LIN {X 0,Y 509.206,Z 475.938,A -85,B 0,C 180,E1 -5494.354,E2 -5494.354} C_VEL
LIN {X 0,Y 509.283,Z 471.955,A -85,B 0,C 180,E1 -5495.543,E2 -5495.543} C_VEL
LIN {X 0,Y 509.306,Z 467.019,A -85,B 0,C 180,E1 -5496.696,E2 -5496.696} C_VEL
LIN {X 0,Y 509.468,Z 461.568,A -85,B 0,C 180,E1 -5497.73,E2 -5497.73} C_VEL
LIN {X 0,Y 509.649,Z 455.252,A -85,B 0,C 180,E1 -5498.725,E2 -5498.725} C_VEL
LIN {X 0,Y 509.834,Z 449.301,A -85,B 0,C 180,E1 -5499.521,E2 -5499.521} C_VEL
LIN {X 0,Y 509.977,Z 442.37,A -85,B 0,C 180,E1 -5500.32,E2 -5500.32} C_VEL
LIN {X 0,Y 510.292,Z 434.19,A -85,B 0,C 180,E1 -5501.117,E2 -5501.117} C_VEL
LIN {X 0,Y 510.576,Z 425.676,A -85,B 0,C 180,E1 -5501.815,E2 -5501.815} C_VEL
LIN {X 0,Y 510.837,Z 415.973,A -85,B 0,C 180,E1 -5502.474,E2 -5502.474} C_VEL
LIN {X 0,Y 511.134,Z 406.186,A -85,B 0,C 180,E1 -5503.012,E2 -5503.012} C_VEL
LIN {X 0,Y 511.34,Z 397.108,A -85,B 0,C 180,E1 -5503.411,E2 -5503.411} C_VEL
LIN {X 0,Y 511.565,Z 387.591,A -85,B 0,C 180,E1 -5503.734,E2 -5503.734} C_VEL
LIN {X 0,Y 511.759,Z 377.276,A -85,B 0,C 180,E1 -5503.982,E2 -5503.982} C_VEL
LIN {X 0,Y 512.077,Z 302.084,A -85,B 0,C 180,E1 -5505.065,E2 -5505.065} C_VEL
LIN {X 0,Y 512.113,Z 283.581,A -85,B 0,C 180,E1 -5505.327,E2 -5505.327} C_VEL
LIN {X 0,Y 510.008,Z 271.254,A -85,B 0,C 180,E1 -5505.588,E2 -5505.588} C_VEL
LIN {X 0,Y 510.017,Z 268.984,A -85,B 0,C 180,E1 -5505.998,E2 -5505.998} C_VEL
LIN {X 0,Y 510.378,Z 255.654,A -85,B 0,C 180,E1 -5508.672,E2 -5508.672} C_VEL
LIN {X 0,Y 510.735,Z 242.059,A -85,B 0,C 180,E1 -5511.386,E2 -5511.386} C_VEL
LIN {X 0,Y 511.204,Z 227.586,A -85,B 0,C 180,E1 -5514.358,E2 -5514.358} C_VEL
LIN {X 0,Y 510.607,Z 222.43,A -85,B 0,C 180,E1 -5515.475,E2 -5515.475} C_VEL
LIN {X 0,Y 509.915,Z 218.493,A -85,B 0,C 180,E1 -5516.407,E2 -5516.407} C_VEL
LIN {X 0,Y 509.86,Z 218.475,A -85,B 0,C 180,E1 -5519.751,E2 -5519.751} C_VEL
LIN {X 0,Y 509.875,Z 218.469,A -85,B 0,C 180,E1 -5522.774,E2 -5522.774} C_VEL
LIN {X 0,Y 509.828,Z 218.476,A -85,B 0,C 180,E1 -5525.578,E2 -5525.578} C_VEL
LIN {X 0,Y 509.852,Z 218.473,A -85,B 0,C 180,E1 -5528.338,E2 -5528.338} C_VEL
LIN {X 0,Y 509.857,Z 218.467,A -85,B 0,C 180,E1 -5531.425,E2 -5531.425} C_VEL
LIN {X 0,Y 509.84,Z 218.472,A -85,B 0,C 180,E1 -5534.67,E2 -5534.67} C_VEL
LIN {X 0,Y 509.835,Z 218.48,A -85,B 0,C 180,E1 -5537.51,E2 -5537.51} C_VEL
LIN {X 0,Y 509.847,Z 218.469,A -85,B 0,C 180,E1 -5540.647,E2 -5540.647} C_VEL
LIN {X 0,Y 509.825,Z 218.479,A -85,B 0,C 180,E1 -5543.646,E2 -5543.646} C_VEL
LIN {X 0,Y 509.842,Z 218.467,A -85,B 0,C 180,E1 -5546.537,E2 -5546.537} C_VEL
LIN {X 0,Y 509.843,Z 218.48,A -85,B 0,C 180,E1 -5549.334,E2 -5549.334} C_VEL
LIN {X 0,Y 509.89,Z 218.461,A -85,B 0,C 180,E1 -5552.054,E2 -5552.054} C_VEL
LIN {X 0,Y 509.876,Z 218.464,A -85,B 0,C 180,E1 -5554.704,E2 -5554.704} C_VEL
LIN {X 0,Y 509.827,Z 218.479,A -85,B 0,C 180,E1 -5557.457,E2 -5557.457} C_VEL
LIN {X 0,Y 509.917,Z 218.457,A -85,B 0,C 180,E1 -5559.844,E2 -5559.844} C_VEL
LIN {X 0,Y 509.872,Z 218.47,A -85,B 0,C 180,E1 -5563.174,E2 -5563.174} C_VEL
LIN {X 0,Y 509.863,Z 218.471,A -85,B 0,C 180,E1 -5565.634,E2 -5565.634} C_VEL
LIN {X 0,Y 509.913,Z 218.465,A -85,B 0,C 180,E1 -5568.874,E2 -5568.874} C_VEL
LIN {X 0,Y 509.921,Z 218.456,A -85,B 0,C 180,E1 -5572.078,E2 -5572.078} C_VEL
LIN {X 0,Y 509.977,Z 218.457,A -85,B 0,C 180,E1 -5574.464,E2 -5574.464} C_VEL
LIN {X 0,Y 510.055,Z 218.443,A -85,B 0,C 180,E1 -5577.63,E2 -5577.63} C_VEL
LIN {X 0,Y 510.063,Z 218.44,A -85,B 0,C 180,E1 -5580.789,E2 -5580.789} C_VEL
LIN {X 0,Y 509.952,Z 218.46,A -85,B 0,C 180,E1 -5583.16,E2 -5583.16} C_VEL
LIN {X 0,Y 509.953,Z 218.462,A -85,B 0,C 180,E1 -5586.329,E2 -5586.329} C_VEL
LIN {X 0,Y 509.914,Z 218.46,A -85,B 0,C 180,E1 -5588.72,E2 -5588.72} C_VEL
LIN {X 0,Y 509.903,Z 218.46,A -85,B 0,C 180,E1 -5591.931,E2 -5591.931} C_VEL
LIN {X 0,Y 509.892,Z 218.466,A -85,B 0,C 180,E1 -5595.241,E2 -5595.241} C_VEL
LIN {X 0,Y 509.887,Z 218.465,A -85,B 0,C 180,E1 -5598,E2 -5598} C_VEL
LIN {X 0,Y 509.848,Z 218.47,A -85,B 0,C 180,E1 -5601.001,E2 -5601.001} C_VEL
LIN {X 0,Y 509.82,Z 218.476,A -85,B 0,C 180,E1 -5603.563,E2 -5603.563} C_VEL
LIN {X 0,Y 509.908,Z 218.462,A -85,B 0,C 180,E1 -5606.378,E2 -5606.378} C_VEL
LIN {X 0,Y 509.873,Z 218.468,A -85,B 0,C 180,E1 -5608.844,E2 -5608.844} C_VEL
LIN {X 0,Y 509.819,Z 218.477,A -85,B 0,C 180,E1 -5611.59,E2 -5611.59} C_VEL
LIN {X 0,Y 509.849,Z 218.471,A -85,B 0,C 180,E1 -5614.413,E2 -5614.413} C_VEL
LIN {X 0,Y 509.816,Z 218.477,A -85,B 0,C 180,E1 -5617.34,E2 -5617.34} C_VEL
LIN {X 0,Y 509.835,Z 218.472,A -85,B 0,C 180,E1 -5620.382,E2 -5620.382} C_VEL
LIN {X 0,Y 509.836,Z 218.473,A -85,B 0,C 180,E1 -5623.064,E2 -5623.064} C_VEL
LIN {X 0,Y 509.828,Z 218.475,A -85,B 0,C 180,E1 -5625.792,E2 -5625.792} C_VEL
LIN {X 0,Y 509.862,Z 218.46,A -85,B 0,C 180,E1 -5628.575,E2 -5628.575} C_VEL
LIN {X 0,Y 509.849,Z 218.48,A -85,B 0,C 180,E1 -5631.786,E2 -5631.786} C_VEL
LIN {X 0,Y 509.827,Z 218.476,A -85,B 0,C 180,E1 -5633.737,E2 -5633.737} C_VEL
LIN {X 0,Y 509.16,Z 218.552,A -85,B 0,C 180,E1 -5634.396,E2 -5634.396} C_VEL
LIN {X 0,Y 506.343,Z 218.904,A -85,B 0,C 180,E1 -5635.468,E2 -5635.468} C_VEL
LIN {X 0,Y 503.951,Z 219.205,A -85,B 0,C 180,E1 -5636.332,E2 -5636.332} C_VEL
LIN {X 0,Y 502.903,Z 219.335,A -85,B 0,C 180,E1 -5636.998,E2 -5636.998} C_VEL
LIN {X 0,Y 502.806,Z 219.347,A -85,B 0,C 180,E1 -5637.224,E2 -5637.224} C_VEL
LIN {X 0,Y 502.811,Z 219.343,A -85,B 0,C 180,E1 -5640.065,E2 -5640.065} C_VEL
LIN {X 0,Y 502.831,Z 219.347,A -85,B 0,C 180,E1 -5642.533,E2 -5642.533} C_VEL
LIN {X 0,Y 502.823,Z 219.354,A -85,B 0,C 180,E1 -5645.299,E2 -5645.299} C_VEL
LIN {X 0,Y 502.776,Z 219.358,A -85,B 0,C 180,E1 -5647.826,E2 -5647.826} C_VEL
LIN {X 0,Y 502.822,Z 219.349,A -85,B 0,C 180,E1 -5650.4,E2 -5650.4} C_VEL
LIN {X 0,Y 502.831,Z 219.351,A -85,B 0,C 180,E1 -5652.932,E2 -5652.932} C_VEL
LIN {X 0,Y 502.848,Z 219.351,A -85,B 0,C 180,E1 -5655.429,E2 -5655.429} C_VEL
LIN {X 0,Y 502.874,Z 219.345,A -85,B 0,C 180,E1 -5658.717,E2 -5658.717} C_VEL
LIN {X 0,Y 502.899,Z 219.341,A -85,B 0,C 180,E1 -5661.967,E2 -5661.967} C_VEL
LIN {X 0,Y 502.939,Z 219.336,A -85,B 0,C 180,E1 -5664.387,E2 -5664.387} C_VEL
LIN {X 0,Y 503.023,Z 219.326,A -85,B 0,C 180,E1 -5667.598,E2 -5667.598} C_VEL
LIN {X 0,Y 503.025,Z 219.325,A -85,B 0,C 180,E1 -5670,E2 -5670} C_VEL
LIN {X 0,Y 503.023,Z 219.326,A -85,B 0,C 180,E1 -5672.402,E2 -5672.402} C_VEL
LIN {X 0,Y 502.939,Z 219.336,A -85,B 0,C 180,E1 -5675.613,E2 -5675.613} C_VEL
LIN {X 0,Y 502.899,Z 219.341,A -85,B 0,C 180,E1 -5678.033,E2 -5678.033} C_VEL
LIN {X 0,Y 502.874,Z 219.345,A -85,B 0,C 180,E1 -5681.283,E2 -5681.283} C_VEL
LIN {X 0,Y 502.848,Z 219.351,A -85,B 0,C 180,E1 -5684.571,E2 -5684.571} C_VEL
LIN {X 0,Y 502.858,Z 219.345,A -85,B 0,C 180,E1 -5687.907,E2 -5687.907} C_VEL
LIN {X 0,Y 502.825,Z 219.355,A -85,B 0,C 180,E1 -5690.536,E2 -5690.536} C_VEL
LIN {X 0,Y 502.788,Z 219.355,A -85,B 0,C 180,E1 -5693.041,E2 -5693.041} C_VEL
LIN {X 0,Y 502.836,Z 219.347,A -85,B 0,C 180,E1 -5695.676,E2 -5695.676} C_VEL
LIN {X 0,Y 502.837,Z 219.347,A -85,B 0,C 180,E1 -5698.373,E2 -5698.373} C_VEL
LIN {X 0,Y 502.793,Z 219.352,A -85,B 0,C 180,E1 -5701.5,E2 -5701.5} C_VEL
LIN {X 0,Y 502.801,Z 219.345,A -85,B 0,C 180,E1 -5704.444,E2 -5704.444} C_VEL
LIN {X 0,Y 502.778,Z 219.353,A -85,B 0,C 180,E1 -5707.179,E2 -5707.179} C_VEL
LIN {X 0,Y 502.818,Z 219.349,A -85,B 0,C 180,E1 -5710.012,E2 -5710.012} C_VEL
LIN {X 0,Y 502.77,Z 219.342,A -85,B 0,C 180,E1 -5713.231,E2 -5713.231} C_VEL
LIN {X 0,Y 502.786,Z 219.352,A -85,B 0,C 180,E1 -5715.662,E2 -5715.662} C_VEL
LIN {X 0,Y 502.83,Z 219.352,A -85,B 0,C 180,E1 -5717.865,E2 -5717.865} C_VEL
LIN {X 0,Y 502.805,Z 219.348,A -85,B 0,C 180,E1 -5721.025,E2 -5721.025} C_VEL
LIN {X 0,Y 502.78,Z 219.352,A -85,B 0,C 180,E1 -5724.168,E2 -5724.168} C_VEL
LIN {X 0,Y 502.83,Z 219.344,A -85,B 0,C 180,E1 -5726.994,E2 -5726.994} C_VEL
LIN {X 0,Y 502.812,Z 219.351,A -85,B 0,C 180,E1 -5730.065,E2 -5730.065} C_VEL
LIN {X 0,Y 502.829,Z 219.337,A -85,B 0,C 180,E1 -5732.534,E2 -5732.534} C_VEL
LIN {X 0,Y 502.783,Z 219.353,A -85,B 0,C 180,E1 -5735.31,E2 -5735.31} C_VEL
LIN {X 0,Y 502.778,Z 219.356,A -85,B 0,C 180,E1 -5737.827,E2 -5737.827} C_VEL
LIN {X 0,Y 502.823,Z 219.337,A -85,B 0,C 180,E1 -5740.401,E2 -5740.401} C_VEL
LIN {X 0,Y 502.832,Z 219.342,A -85,B 0,C 180,E1 -5742.932,E2 -5742.932} C_VEL
LIN {X 0,Y 502.85,Z 219.351,A -85,B 0,C 180,E1 -5745.43,E2 -5745.43} C_VEL
LIN {X 0,Y 502.876,Z 219.335,A -85,B 0,C 180,E1 -5748.717,E2 -5748.717} C_VEL
LIN {X 0,Y 502.901,Z 219.335,A -85,B 0,C 180,E1 -5751.967,E2 -5751.967} C_VEL
LIN {X 0,Y 502.933,Z 219.333,A -85,B 0,C 180,E1 -5754.387,E2 -5754.387} C_VEL
LIN {X 0,Y 503.025,Z 219.319,A -85,B 0,C 180,E1 -5757.598,E2 -5757.598} C_VEL
LIN {X 0,Y 503.027,Z 219.31,A -85,B 0,C 180,E1 -5760,E2 -5760} C_VEL
LIN {X 0,Y 503.024,Z 219.318,A -85,B 0,C 180,E1 -5762.403,E2 -5762.403} C_VEL
LIN {X 0,Y 502.93,Z 219.334,A -85,B 0,C 180,E1 -5765.614,E2 -5765.614} C_VEL
LIN {X 0,Y 502.864,Z 219.338,A -85,B 0,C 180,E1 -5768.844,E2 -5768.844} C_VEL
LIN {X 0,Y 502.846,Z 219.34,A -85,B 0,C 180,E1 -5772.102,E2 -5772.102} C_VEL
LIN {X 0,Y 502.849,Z 219.343,A -85,B 0,C 180,E1 -5775.4,E2 -5775.4} C_VEL
LIN {X 0,Y 502.826,Z 219.342,A -85,B 0,C 180,E1 -5778.752,E2 -5778.752} C_VEL
LIN {X 0,Y 502.783,Z 219.352,A -85,B 0,C 180,E1 -5781.312,E2 -5781.312} C_VEL
LIN {X 0,Y 502.785,Z 219.351,A -85,B 0,C 180,E1 -5783.914,E2 -5783.914} C_VEL
LIN {X 0,Y 502.865,Z 219.34,A -85,B 0,C 180,E1 -5786.566,E2 -5786.566} C_VEL
LIN {X 0,Y 502.824,Z 219.347,A -85,B 0,C 180,E1 -5789.288,E2 -5789.288} C_VEL
LIN {X 0,Y 502.782,Z 219.354,A -85,B 0,C 180,E1 -5792.085,E2 -5792.085} C_VEL
LIN {X 0,Y 502.796,Z 219.35,A -85,B 0,C 180,E1 -5794.966,E2 -5794.966} C_VEL
LIN {X 0,Y 502.794,Z 219.353,A -85,B 0,C 180,E1 -5797.954,E2 -5797.954} C_VEL
LIN {X 0,Y 502.821,Z 219.347,A -85,B 0,C 180,E1 -5801.066,E2 -5801.066} C_VEL
LIN {X 0,Y 502.787,Z 219.355,A -85,B 0,C 180,E1 -5804.53,E2 -5804.53} C_VEL
LIN {X 0,Y 502.797,Z 219.354,A -85,B 0,C 180,E1 -5807.861,E2 -5807.861} C_VEL
LIN {X 0,Y 502.804,Z 219.349,A -85,B 0,C 180,E1 -5811.024,E2 -5811.024} C_VEL
LIN {X 0,Y 502.777,Z 219.354,A -85,B 0,C 180,E1 -5814.169,E2 -5814.169} C_VEL
LIN {X 0,Y 502.835,Z 219.345,A -85,B 0,C 180,E1 -5816.994,E2 -5816.994} C_VEL
LIN {X 0,Y 502.817,Z 219.352,A -85,B 0,C 180,E1 -5820.065,E2 -5820.065} C_VEL
LIN {X 0,Y 502.878,Z 219.516,A -85,B 0,C 180,E1 -5823.479,E2 -5823.479} C_VEL
LIN {X 0,Y 504.2,Z 227.447,A -85,B 0,C 180,E1 -5825.281,E2 -5825.281} C_VEL
LIN {X 0,Y 503.846,Z 238.784,A -85,B 0,C 180,E1 -5827.66,E2 -5827.66} C_VEL
LIN {X 0,Y 503.534,Z 251.309,A -85,B 0,C 180,E1 -5830.217,E2 -5830.217} C_VEL
LIN {X 0,Y 503.109,Z 265.765,A -85,B 0,C 180,E1 -5833.151,E2 -5833.151} C_VEL
LIN {X 0,Y 502.954,Z 270.794,A -85,B 0,C 180,E1 -5834.165,E2 -5834.165} C_VEL
LIN {X 0,Y 503.729,Z 275.59,A -85,B 0,C 180,E1 -5834.3,E2 -5834.3} C_VEL
LIN {X 0,Y 505.349,Z 285.243,A -85,B 0,C 180,E1 -5834.49,E2 -5834.49} C_VEL
LIN {X 0,Y 504.877,Z 375.752,A -85,B 0,C 180,E1 -5835.798,E2 -5835.798} C_VEL
LIN {X 0,Y 504.677,Z 386.523,A -85,B 0,C 180,E1 -5836.049,E2 -5836.049} C_VEL
LIN {X 0,Y 504.465,Z 395.627,A -85,B 0,C 180,E1 -5836.351,E2 -5836.351} C_VEL
LIN {X 0,Y 504.192,Z 405.993,A -85,B 0,C 180,E1 -5836.806,E2 -5836.806} C_VEL
LIN {X 0,Y 503.889,Z 415.953,A -85,B 0,C 180,E1 -5837.362,E2 -5837.362} C_VEL
LIN {X 0,Y 503.605,Z 424.129,A -85,B 0,C 180,E1 -5837.917,E2 -5837.917} C_VEL
LIN {X 0,Y 503.336,Z 432.861,A -85,B 0,C 180,E1 -5838.625,E2 -5838.625} C_VEL
LIN {X 0,Y 503.048,Z 440.257,A -85,B 0,C 180,E1 -5839.332,E2 -5839.332} C_VEL
LIN {X 0,Y 502.842,Z 447.479,A -85,B 0,C 180,E1 -5840.142,E2 -5840.142} C_VEL
LIN {X 0,Y 502.642,Z 453.682,A -85,B 0,C 180,E1 -5840.95,E2 -5840.95} C_VEL
LIN {X 0,Y 502.437,Z 460.219,A -85,B 0,C 180,E1 -5841.959,E2 -5841.959} C_VEL
LIN {X 0,Y 502.275,Z 465.773,A -85,B 0,C 180,E1 -5842.988,E2 -5842.988} C_VEL
LIN {X 0,Y 502.201,Z 470.209,A -85,B 0,C 180,E1 -5843.975,E2 -5843.975} C_VEL
LIN {X 0,Y 502.112,Z 474.529,A -85,B 0,C 180,E1 -5845.183,E2 -5845.183} C_VEL
LIN {X 0,Y 502.139,Z 476.894,A -85,B 0,C 180,E1 -5845.987,E2 -5845.987} C_VEL
LIN {X 0,Y 502.12,Z 478.689,A -85,B 0,C 180,E1 -5846.791,E2 -5846.791} C_VEL
LIN {X 0,Y 502.037,Z 481.127,A -85,B 0,C 180,E1 -5848.396,E2 -5848.396} C_VEL
LIN {X 0,Y 501.991,Z 481.713,A -85,B 0,C 180,E1 -5849.198,E2 -5849.198} C_VEL
LIN {X 0,Y 501.991,Z 481.713,A -85,B 0,C 180,E1 -5850.802,E2 -5850.802} C_VEL
LIN {X 0,Y 502.037,Z 481.127,A -85,B 0,C 180,E1 -5851.604,E2 -5851.604} C_VEL
LIN {X 0,Y 502.12,Z 478.689,A -85,B 0,C 180,E1 -5853.209,E2 -5853.209} C_VEL
LIN {X 0,Y 502.105,Z 475.744,A -85,B 0,C 180,E1 -5854.415,E2 -5854.415} C_VEL
LIN {X 0,Y 502.199,Z 471.762,A -85,B 0,C 180,E1 -5855.622,E2 -5855.622} C_VEL
LIN {X 0,Y 502.219,Z 466.825,A -85,B 0,C 180,E1 -5856.791,E2 -5856.791} C_VEL
LIN {X 0,Y 502.393,Z 461.374,A -85,B 0,C 180,E1 -5857.839,E2 -5857.839} C_VEL
LIN {X 0,Y 502.59,Z 455.058,A -85,B 0,C 180,E1 -5858.848,E2 -5858.848} C_VEL
LIN {X 0,Y 502.796,Z 449.107,A -85,B 0,C 180,E1 -5859.656,E2 -5859.656} C_VEL
LIN {X 0,Y 502.954,Z 442.176,A -85,B 0,C 180,E1 -5860.466,E2 -5860.466} C_VEL
LIN {X 0,Y 503.289,Z 433.996,A -85,B 0,C 180,E1 -5861.274,E2 -5861.274} C_VEL
LIN {X 0,Y 503.601,Z 425.482,A -85,B 0,C 180,E1 -5861.981,E2 -5861.981} C_VEL
LIN {X 0,Y 503.869,Z 416.244,A -85,B 0,C 180,E1 -5862.62,E2 -5862.62} C_VEL
LIN {X 0,Y 504.182,Z 407,A -85,B 0,C 180,E1 -5863.143,E2 -5863.143} C_VEL
LIN {X 0,Y 504.423,Z 396.915,A -85,B 0,C 180,E1 -5863.598,E2 -5863.598} C_VEL
LIN {X 0,Y 504.675,Z 387.398,A -85,B 0,C 180,E1 -5863.925,E2 -5863.925} C_VEL
LIN {X 0,Y 504.888,Z 377.084,A -85,B 0,C 180,E1 -5864.176,E2 -5864.176} C_VEL
LIN {X 0,Y 505.229,Z 303.681,A -85,B 0,C 180,E1 -5865.248,E2 -5865.248} C_VEL
LIN {X 0,Y 505.146,Z 283.952,A -85,B 0,C 180,E1 -5865.535,E2 -5865.535} C_VEL
LIN {X 0,Y 502.987,Z 271.213,A -85,B 0,C 180,E1 -5865.803,E2 -5865.803} C_VEL
LIN {X 0,Y 502.955,Z 270.102,A -85,B 0,C 180,E1 -5865.947,E2 -5865.947} C_VEL
LIN {X 0,Y 503.374,Z 256.567,A -85,B 0,C 180,E1 -5868.731,E2 -5868.731} C_VEL
LIN {X 0,Y 503.759,Z 242.972,A -85,B 0,C 180,E1 -5871.482,E2 -5871.482} C_VEL
LIN {X 0,Y 504.242,Z 228.511,A -85,B 0,C 180,E1 -5874.497,E2 -5874.497} C_VEL
LIN {X 0,Y 503.202,Z 221.288,A -85,B 0,C 180,E1 -5876.1,E2 -5876.1} C_VEL
LIN {X 0,Y 502.852,Z 219.371,A -85,B 0,C 180,E1 -5876.595,E2 -5876.595} C_VEL
LIN {X 0,Y 502.817,Z 219.352,A -85,B 0,C 180,E1 -5879.935,E2 -5879.935} C_VEL
LIN {X 0,Y 502.834,Z 219.346,A -85,B 0,C 180,E1 -5883.031,E2 -5883.031} C_VEL
LIN {X 0,Y 502.775,Z 219.354,A -85,B 0,C 180,E1 -5885.951,E2 -5885.951} C_VEL
LIN {X 0,Y 502.804,Z 219.349,A -85,B 0,C 180,E1 -5888.976,E2 -5888.976} C_VEL
LIN {X 0,Y 502.797,Z 219.353,A -85,B 0,C 180,E1 -5892.139,E2 -5892.139} C_VEL
LIN {X 0,Y 502.787,Z 219.355,A -85,B 0,C 180,E1 -5895.47,E2 -5895.47} C_VEL
LIN {X 0,Y 502.821,Z 219.347,A -85,B 0,C 180,E1 -5898.934,E2 -5898.934} C_VEL
LIN {X 0,Y 502.794,Z 219.353,A -85,B 0,C 180,E1 -5902.046,E2 -5902.046} C_VEL
LIN {X 0,Y 502.796,Z 219.35,A -85,B 0,C 180,E1 -5905.033,E2 -5905.033} C_VEL
LIN {X 0,Y 502.782,Z 219.354,A -85,B 0,C 180,E1 -5907.915,E2 -5907.915} C_VEL
LIN {X 0,Y 502.824,Z 219.347,A -85,B 0,C 180,E1 -5910.712,E2 -5910.712} C_VEL
LIN {X 0,Y 502.863,Z 219.34,A -85,B 0,C 180,E1 -5913.439,E2 -5913.439} C_VEL
LIN {X 0,Y 502.785,Z 219.351,A -85,B 0,C 180,E1 -5916.086,E2 -5916.086} C_VEL
LIN {X 0,Y 502.783,Z 219.352,A -85,B 0,C 180,E1 -5918.688,E2 -5918.688} C_VEL
LIN {X 0,Y 502.826,Z 219.342,A -85,B 0,C 180,E1 -5921.248,E2 -5921.248} C_VEL
LIN {X 0,Y 502.849,Z 219.343,A -85,B 0,C 180,E1 -5924.6,E2 -5924.6} C_VEL
LIN {X 0,Y 502.876,Z 219.336,A -85,B 0,C 180,E1 -5928.039,E2 -5928.039} C_VEL
LIN {X 0,Y 502.864,Z 219.338,A -85,B 0,C 180,E1 -5931.156,E2 -5931.156} C_VEL
LIN {X 0,Y 502.93,Z 219.334,A -85,B 0,C 180,E1 -5934.386,E2 -5934.386} C_VEL
LIN {X 0,Y 503.024,Z 219.318,A -85,B 0,C 180,E1 -5937.597,E2 -5937.597} C_VEL
LIN {X 0,Y 503.027,Z 219.31,A -85,B 0,C 180,E1 -5940,E2 -5940} C_VEL
LIN {X 0,Y 503.025,Z 219.319,A -85,B 0,C 180,E1 -5942.402,E2 -5942.402} C_VEL
LIN {X 0,Y 502.933,Z 219.333,A -85,B 0,C 180,E1 -5945.613,E2 -5945.613} C_VEL
LIN {X 0,Y 502.901,Z 219.335,A -85,B 0,C 180,E1 -5948.033,E2 -5948.033} C_VEL
LIN {X 0,Y 502.876,Z 219.335,A -85,B 0,C 180,E1 -5951.283,E2 -5951.283} C_VEL
LIN {X 0,Y 502.85,Z 219.351,A -85,B 0,C 180,E1 -5954.57,E2 -5954.57} C_VEL
LIN {X 0,Y 502.86,Z 219.339,A -85,B 0,C 180,E1 -5957.907,E2 -5957.907} C_VEL
LIN {X 0,Y 502.827,Z 219.348,A -85,B 0,C 180,E1 -5960.536,E2 -5960.536} C_VEL
LIN {X 0,Y 502.786,Z 219.352,A -85,B 0,C 180,E1 -5963.04,E2 -5963.04} C_VEL
LIN {X 0,Y 502.819,Z 219.346,A -85,B 0,C 180,E1 -5965.676,E2 -5965.676} C_VEL
LIN {X 0,Y 502.837,Z 219.347,A -85,B 0,C 180,E1 -5968.372,E2 -5968.372} C_VEL
LIN {X 0,Y 502.791,Z 219.352,A -85,B 0,C 180,E1 -5971.499,E2 -5971.499} C_VEL
LIN {X 0,Y 502.801,Z 219.348,A -85,B 0,C 180,E1 -5974.444,E2 -5974.444} C_VEL
LIN {X 0,Y 502.778,Z 219.353,A -85,B 0,C 180,E1 -5977.178,E2 -5977.178} C_VEL
LIN {X 0,Y 502.785,Z 219.354,A -85,B 0,C 180,E1 -5980.015,E2 -5980.015} C_VEL
LIN {X 0,Y 502.818,Z 219.353,A -85,B 0,C 180,E1 -5982.201,E2 -5982.201} C_VEL
LIN {X 0,Y 502.797,Z 219.351,A -85,B 0,C 180,E1 -5985.468,E2 -5985.468} C_VEL
LIN {X 0,Y 502.823,Z 219.336,A -85,B 0,C 180,E1 -5989.004,E2 -5989.004} C_VEL
LIN {X 0,Y 502.791,Z 219.356,A -85,B 0,C 180,E1 -5992.046,E2 -5992.046} C_VEL
LIN {X 0,Y 502.803,Z 219.343,A -85,B 0,C 180,E1 -5995.035,E2 -5995.035} C_VEL
LIN {X 0,Y 502.806,Z 219.347,A -85,B 0,C 180,E1 -5997.224,E2 -5997.224} C_VEL
LIN {X 0,Y 502.106,Z 219.442,A -85,B 0,C 180,E1 -5997.892,E2 -5997.892} C_VEL
LIN {X 0,Y 499.24,Z 219.795,A -85,B 0,C 180,E1 -5998.978,E2 -5998.978} C_VEL
LIN {X 0,Y 496.845,Z 220.089,A -85,B 0,C 180,E1 -5999.853,E2 -5999.853} C_VEL
LIN {X 0,Y 495.827,Z 220.211,A -85,B 0,C 180,E1 -6000.529,E2 -6000.529} C_VEL
LIN {X 0,Y 495.749,Z 220.22,A -85,B 0,C 180,E1 -6000.757,E2 -6000.757} C_VEL
LIN {X 0,Y 495.787,Z 220.228,A -85,B 0,C 180,E1 -6003.932,E2 -6003.932} C_VEL
LIN {X 0,Y 495.756,Z 220.233,A -85,B 0,C 180,E1 -6007.139,E2 -6007.139} C_VEL
LIN {X 0,Y 495.774,Z 220.228,A -85,B 0,C 180,E1 -6010.11,E2 -6010.11} C_VEL
LIN {X 0,Y 495.783,Z 220.227,A -85,B 0,C 180,E1 -6012.681,E2 -6012.681} C_VEL
LIN {X 0,Y 495.791,Z 220.231,A -85,B 0,C 180,E1 -6015.217,E2 -6015.217} C_VEL
LIN {X 0,Y 495.849,Z 220.219,A -85,B 0,C 180,E1 -6018.555,E2 -6018.555} C_VEL
LIN {X 0,Y 495.87,Z 220.217,A -85,B 0,C 180,E1 -6021.852,E2 -6021.852} C_VEL
LIN {X 0,Y 495.897,Z 220.213,A -85,B 0,C 180,E1 -6024.307,E2 -6024.307} C_VEL
LIN {X 0,Y 495.992,Z 220.203,A -85,B 0,C 180,E1 -6027.564,E2 -6027.564} C_VEL
LIN {X 0,Y 495.996,Z 220.2,A -85,B 0,C 180,E1 -6030,E2 -6030} C_VEL
LIN {X 0,Y 495.992,Z 220.202,A -85,B 0,C 180,E1 -6032.436,E2 -6032.436} C_VEL
LIN {X 0,Y 495.897,Z 220.213,A -85,B 0,C 180,E1 -6035.693,E2 -6035.693} C_VEL
LIN {X 0,Y 495.87,Z 220.217,A -85,B 0,C 180,E1 -6038.148,E2 -6038.148} C_VEL
LIN {X 0,Y 495.849,Z 220.219,A -85,B 0,C 180,E1 -6041.445,E2 -6041.445} C_VEL
LIN {X 0,Y 495.791,Z 220.231,A -85,B 0,C 180,E1 -6044.783,E2 -6044.783} C_VEL
LIN {X 0,Y 495.783,Z 220.227,A -85,B 0,C 180,E1 -6047.319,E2 -6047.319} C_VEL
LIN {X 0,Y 495.774,Z 220.228,A -85,B 0,C 180,E1 -6049.89,E2 -6049.89} C_VEL
LIN {X 0,Y 495.756,Z 220.233,A -85,B 0,C 180,E1 -6052.861,E2 -6052.861} C_VEL
LIN {X 0,Y 495.787,Z 220.228,A -85,B 0,C 180,E1 -6056.068,E2 -6056.068} C_VEL
LIN {X 0,Y 495.768,Z 220.22,A -85,B 0,C 180,E1 -6058.815,E2 -6058.815} C_VEL
LIN {X 0,Y 495.755,Z 220.229,A -85,B 0,C 180,E1 -6061.726,E2 -6061.726} C_VEL
LIN {X 0,Y 495.771,Z 220.219,A -85,B 0,C 180,E1 -6064.695,E2 -6064.695} C_VEL
LIN {X 0,Y 495.728,Z 220.232,A -85,B 0,C 180,E1 -6067.562,E2 -6067.562} C_VEL
LIN {X 0,Y 495.776,Z 220.215,A -85,B 0,C 180,E1 -6070.699,E2 -6070.699} C_VEL
LIN {X 0,Y 495.731,Z 220.226,A -85,B 0,C 180,E1 -6074.001,E2 -6074.001} C_VEL
LIN {X 0,Y 495.759,Z 220.227,A -85,B 0,C 180,E1 -6077.121,E2 -6077.121} C_VEL
LIN {X 0,Y 495.777,Z 220.227,A -85,B 0,C 180,E1 -6080.365,E2 -6080.365} C_VEL
LIN {X 0,Y 495.73,Z 220.233,A -85,B 0,C 180,E1 -6083.457,E2 -6083.457} C_VEL
LIN {X 0,Y 495.757,Z 220.226,A -85,B 0,C 180,E1 -6086.436,E2 -6086.436} C_VEL
LIN {X 0,Y 495.749,Z 220.231,A -85,B 0,C 180,E1 -6089.313,E2 -6089.313} C_VEL
LIN {X 0,Y 495.777,Z 220.218,A -85,B 0,C 180,E1 -6092.109,E2 -6092.109} C_VEL
LIN {X 0,Y 495.75,Z 220.226,A -85,B 0,C 180,E1 -6094.831,E2 -6094.831} C_VEL
LIN {X 0,Y 495.746,Z 220.235,A -85,B 0,C 180,E1 -6097.495,E2 -6097.495} C_VEL
LIN {X 0,Y 495.769,Z 220.216,A -85,B 0,C 180,E1 -6100.11,E2 -6100.11} C_VEL
LIN {X 0,Y 495.784,Z 220.219,A -85,B 0,C 180,E1 -6102.682,E2 -6102.682} C_VEL
LIN {X 0,Y 495.793,Z 220.227,A -85,B 0,C 180,E1 -6105.218,E2 -6105.218} C_VEL
LIN {X 0,Y 495.85,Z 220.209,A -85,B 0,C 180,E1 -6108.555,E2 -6108.555} C_VEL
LIN {X 0,Y 495.872,Z 220.211,A -85,B 0,C 180,E1 -6111.853,E2 -6111.853} C_VEL
LIN {X 0,Y 495.889,Z 220.21,A -85,B 0,C 180,E1 -6114.307,E2 -6114.307} C_VEL
LIN {X 0,Y 495.993,Z 220.195,A -85,B 0,C 180,E1 -6117.564,E2 -6117.564} C_VEL
LIN {X 0,Y 495.982,Z 220.19,A -85,B 0,C 180,E1 -6120.812,E2 -6120.812} C_VEL
LIN {X 0,Y 495.993,Z 220.194,A -85,B 0,C 180,E1 -6122.437,E2 -6122.437} C_VEL
LIN {X 0,Y 495.885,Z 220.211,A -85,B 0,C 180,E1 -6125.694,E2 -6125.694} C_VEL
LIN {X 0,Y 495.834,Z 220.211,A -85,B 0,C 180,E1 -6128.97,E2 -6128.97} C_VEL
LIN {X 0,Y 495.828,Z 220.214,A -85,B 0,C 180,E1 -6132.035,E2 -6132.035} C_VEL
LIN {X 0,Y 495.824,Z 220.218,A -85,B 0,C 180,E1 -6135.452,E2 -6135.452} C_VEL
LIN {X 0,Y 495.778,Z 220.216,A -85,B 0,C 180,E1 -6138.238,E2 -6138.238} C_VEL
LIN {X 0,Y 495.774,Z 220.226,A -85,B 0,C 180,E1 -6140.757,E2 -6140.757} C_VEL
LIN {X 0,Y 495.748,Z 220.228,A -85,B 0,C 180,E1 -6143.388,E2 -6143.388} C_VEL
LIN {X 0,Y 495.791,Z 220.218,A -85,B 0,C 180,E1 -6146.068,E2 -6146.068} C_VEL
LIN {X 0,Y 495.772,Z 220.23,A -85,B 0,C 180,E1 -6148.815,E2 -6148.815} C_VEL
LIN {X 0,Y 495.755,Z 220.227,A -85,B 0,C 180,E1 -6151.725,E2 -6151.725} C_VEL
LIN {X 0,Y 495.763,Z 220.228,A -85,B 0,C 180,E1 -6154.693,E2 -6154.693} C_VEL
LIN {X 0,Y 495.73,Z 220.231,A -85,B 0,C 180,E1 -6157.562,E2 -6157.562} C_VEL
LIN {X 0,Y 495.767,Z 220.229,A -85,B 0,C 180,E1 -6160.7,E2 -6160.7} C_VEL
LIN {X 0,Y 495.73,Z 220.234,A -85,B 0,C 180,E1 -6164.002,E2 -6164.002} C_VEL
LIN {X 0,Y 495.727,Z 220.231,A -85,B 0,C 180,E1 -6167.117,E2 -6167.117} C_VEL
LIN {X 0,Y 495.761,Z 220.222,A -85,B 0,C 180,E1 -6169.953,E2 -6169.953} C_VEL
LIN {X 0,Y 495.73,Z 220.233,A -85,B 0,C 180,E1 -6172.554,E2 -6172.554} C_VEL
LIN {X 0,Y 495.78,Z 220.225,A -85,B 0,C 180,E1 -6175.457,E2 -6175.457} C_VEL
LIN {X 0,Y 495.758,Z 220.234,A -85,B 0,C 180,E1 -6178.364,E2 -6178.364} C_VEL
LIN {X 0,Y 495.758,Z 220.234,A -85,B 0,C 180,E1 -6181.514,E2 -6181.514} C_VEL
LIN {X 0,Y 495.846,Z 220.414,A -85,B 0,C 180,E1 -6183.297,E2 -6183.297} C_VEL
LIN {X 0,Y 497.275,Z 229.398,A -85,B 0,C 180,E1 -6185.36,E2 -6185.36} C_VEL
LIN {X 0,Y 496.788,Z 243.885,A -85,B 0,C 180,E1 -6188.419,E2 -6188.419} C_VEL
LIN {X 0,Y 496.338,Z 258.026,A -85,B 0,C 180,E1 -6191.35,E2 -6191.35} C_VEL
LIN {X 0,Y 495.952,Z 270.636,A -85,B 0,C 180,E1 -6193.938,E2 -6193.938} C_VEL
LIN {X 0,Y 496.776,Z 275.595,A -85,B 0,C 180,E1 -6194.077,E2 -6194.077} C_VEL
LIN {X 0,Y 498.494,Z 286.293,A -85,B 0,C 180,E1 -6194.289,E2 -6194.289} C_VEL
LIN {X 0,Y 497.997,Z 375.559,A -85,B 0,C 180,E1 -6195.598,E2 -6195.598} C_VEL
LIN {X 0,Y 497.782,Z 386.33,A -85,B 0,C 180,E1 -6195.852,E2 -6195.852} C_VEL
LIN {X 0,Y 497.555,Z 395.434,A -85,B 0,C 180,E1 -6196.158,E2 -6196.158} C_VEL
LIN {X 0,Y 497.274,Z 405.8,A -85,B 0,C 180,E1 -6196.619,E2 -6196.619} C_VEL
LIN {X 0,Y 496.974,Z 414.976,A -85,B 0,C 180,E1 -6197.133,E2 -6197.133} C_VEL
LIN {X 0,Y 496.649,Z 423.936,A -85,B 0,C 180,E1 -6197.745,E2 -6197.745} C_VEL
LIN {X 0,Y 496.371,Z 432.668,A -85,B 0,C 180,E1 -6198.464,E2 -6198.464} C_VEL
LIN {X 0,Y 496.059,Z 440.064,A -85,B 0,C 180,E1 -6199.18,E2 -6199.18} C_VEL
LIN {X 0,Y 495.813,Z 447.286,A -85,B 0,C 180,E1 -6200.001,E2 -6200.001} C_VEL
LIN {X 0,Y 495.608,Z 453.489,A -85,B 0,C 180,E1 -6200.82,E2 -6200.82} C_VEL
LIN {X 0,Y 495.384,Z 460.026,A -85,B 0,C 180,E1 -6201.844,E2 -6201.844} C_VEL
LIN {X 0,Y 495.263,Z 464.527,A -85,B 0,C 180,E1 -6202.663,E2 -6202.663} C_VEL
LIN {X 0,Y 495.118,Z 469.552,A -85,B 0,C 180,E1 -6203.767,E2 -6203.767} C_VEL
LIN {X 0,Y 495.104,Z 473.098,A -85,B 0,C 180,E1 -6204.706,E2 -6204.706} C_VEL
LIN {X 0,Y 495.033,Z 476.7,A -85,B 0,C 180,E1 -6205.929,E2 -6205.929} C_VEL
LIN {X 0,Y 495.042,Z 478.497,A -85,B 0,C 180,E1 -6206.745,E2 -6206.745} C_VEL
LIN {X 0,Y 494.963,Z 480.935,A -85,B 0,C 180,E1 -6208.373,E2 -6208.373} C_VEL
LIN {X 0,Y 494.911,Z 481.521,A -85,B 0,C 180,E1 -6209.186,E2 -6209.186} C_VEL
LIN {X 0,Y 494.911,Z 481.521,A -85,B 0,C 180,E1 -6210.814,E2 -6210.814} C_VEL
LIN {X 0,Y 494.963,Z 480.935,A -85,B 0,C 180,E1 -6211.627,E2 -6211.627} C_VEL
LIN {X 0,Y 495.042,Z 478.497,A -85,B 0,C 180,E1 -6213.255,E2 -6213.255} C_VEL
LIN {X 0,Y 495.01,Z 475.551,A -85,B 0,C 180,E1 -6214.479,E2 -6214.479} C_VEL
LIN {X 0,Y 495.116,Z 471.569,A -85,B 0,C 180,E1 -6215.702,E2 -6215.702} C_VEL
LIN {X 0,Y 495.169,Z 466.441,A -85,B 0,C 180,E1 -6216.929,E2 -6216.929} C_VEL
LIN {X 0,Y 495.338,Z 461.181,A -85,B 0,C 180,E1 -6217.952,E2 -6217.952} C_VEL
LIN {X 0,Y 495.556,Z 454.865,A -85,B 0,C 180,E1 -6218.975,E2 -6218.975} C_VEL
LIN {X 0,Y 495.747,Z 448.913,A -85,B 0,C 180,E1 -6219.795,E2 -6219.795} C_VEL
LIN {X 0,Y 495.953,Z 441.983,A -85,B 0,C 180,E1 -6220.616,E2 -6220.616} C_VEL
LIN {X 0,Y 496.304,Z 433.802,A -85,B 0,C 180,E1 -6221.435,E2 -6221.435} C_VEL
LIN {X 0,Y 496.622,Z 425.288,A -85,B 0,C 180,E1 -6222.152,E2 -6222.152} C_VEL
LIN {X 0,Y 496.906,Z 416.521,A -85,B 0,C 180,E1 -6222.77,E2 -6222.77} C_VEL
LIN {X 0,Y 497.28,Z 406.808,A -85,B 0,C 180,E1 -6223.329,E2 -6223.329} C_VEL
LIN {X 0,Y 497.513,Z 396.721,A -85,B 0,C 180,E1 -6223.791,E2 -6223.791} C_VEL
LIN {X 0,Y 497.778,Z 387.205,A -85,B 0,C 180,E1 -6224.122,E2 -6224.122} C_VEL
LIN {X 0,Y 498.022,Z 376.892,A -85,B 0,C 180,E1 -6224.376,E2 -6224.376} C_VEL
LIN {X 0,Y 498.37,Z 303.21,A -85,B 0,C 180,E1 -6225.467,E2 -6225.467} C_VEL
LIN {X 0,Y 498.337,Z 285.015,A -85,B 0,C 180,E1 -6225.734,E2 -6225.734} C_VEL
LIN {X 0,Y 495.954,Z 270.875,A -85,B 0,C 180,E1 -6226.042,E2 -6226.042} C_VEL
LIN {X 0,Y 495.964,Z 269.579,A -85,B 0,C 180,E1 -6226.252,E2 -6226.252} C_VEL
LIN {X 0,Y 496.377,Z 258.143,A -85,B 0,C 180,E1 -6228.655,E2 -6228.655} C_VEL
LIN {X 0,Y 496.779,Z 243.885,A -85,B 0,C 180,E1 -6231.581,E2 -6231.581} C_VEL
LIN {X 0,Y 497.286,Z 230.46,A -85,B 0,C 180,E1 -6234.417,E2 -6234.417} C_VEL
LIN {X 0,Y 496.733,Z 225.312,A -85,B 0,C 180,E1 -6235.564,E2 -6235.564} C_VEL
LIN {X 0,Y 495.796,Z 220.251,A -85,B 0,C 180,E1 -6236.78,E2 -6236.78} C_VEL
LIN {X 0,Y 495.767,Z 220.231,A -85,B 0,C 180,E1 -6240.147,E2 -6240.147} C_VEL
LIN {X 0,Y 495.795,Z 220.223,A -85,B 0,C 180,E1 -6243.244,E2 -6243.244} C_VEL
LIN {X 0,Y 495.721,Z 220.234,A -85,B 0,C 180,E1 -6246.088,E2 -6246.088} C_VEL
LIN {X 0,Y 495.765,Z 220.225,A -85,B 0,C 180,E1 -6248.768,E2 -6248.768} C_VEL
LIN {X 0,Y 495.758,Z 220.227,A -85,B 0,C 180,E1 -6251.781,E2 -6251.781} C_VEL
LIN {X 0,Y 495.739,Z 220.23,A -85,B 0,C 180,E1 -6255.14,E2 -6255.14} C_VEL
LIN {X 0,Y 495.757,Z 220.228,A -85,B 0,C 180,E1 -6258.219,E2 -6258.219} C_VEL
LIN {X 0,Y 495.751,Z 220.23,A -85,B 0,C 180,E1 -6261.408,E2 -6261.408} C_VEL
LIN {X 0,Y 495.747,Z 220.226,A -85,B 0,C 180,E1 -6264.462,E2 -6264.462} C_VEL
LIN {X 0,Y 495.752,Z 220.23,A -85,B 0,C 180,E1 -6267.404,E2 -6267.404} C_VEL
LIN {X 0,Y 495.766,Z 220.225,A -85,B 0,C 180,E1 -6270.253,E2 -6270.253} C_VEL
LIN {X 0,Y 495.824,Z 220.215,A -85,B 0,C 180,E1 -6273.25,E2 -6273.25} C_VEL
LIN {X 0,Y 495.748,Z 220.23,A -85,B 0,C 180,E1 -6275.724,E2 -6275.724} C_VEL
LIN {X 0,Y 495.743,Z 220.227,A -85,B 0,C 180,E1 -6278.371,E2 -6278.371} C_VEL
LIN {X 0,Y 495.782,Z 220.22,A -85,B 0,C 180,E1 -6280.971,E2 -6280.971} C_VEL
LIN {X 0,Y 495.807,Z 220.219,A -85,B 0,C 180,E1 -6284.376,E2 -6284.376} C_VEL
LIN {X 0,Y 495.783,Z 220.229,A -85,B 0,C 180,E1 -6286.89,E2 -6286.89} C_VEL
LIN {X 0,Y 495.773,Z 220.216,A -85,B 0,C 180,E1 -6289.38,E2 -6289.38} C_VEL
LIN {X 0,Y 495.836,Z 220.21,A -85,B 0,C 180,E1 -6291.851,E2 -6291.851} C_VEL
LIN {X 0,Y 495.885,Z 220.211,A -85,B 0,C 180,E1 -6294.306,E2 -6294.306} C_VEL
LIN {X 0,Y 495.993,Z 220.194,A -85,B 0,C 180,E1 -6297.563,E2 -6297.563} C_VEL
LIN {X 0,Y 495.983,Z 220.192,A -85,B 0,C 180,E1 -6300.811,E2 -6300.811} C_VEL
LIN {X 0,Y 495.993,Z 220.195,A -85,B 0,C 180,E1 -6302.436,E2 -6302.436} C_VEL
LIN {X 0,Y 495.889,Z 220.21,A -85,B 0,C 180,E1 -6305.693,E2 -6305.693} C_VEL
LIN {X 0,Y 495.872,Z 220.211,A -85,B 0,C 180,E1 -6308.147,E2 -6308.147} C_VEL
LIN {X 0,Y 495.85,Z 220.209,A -85,B 0,C 180,E1 -6311.445,E2 -6311.445} C_VEL
LIN {X 0,Y 495.793,Z 220.227,A -85,B 0,C 180,E1 -6314.782,E2 -6314.782} C_VEL
LIN {X 0,Y 495.784,Z 220.219,A -85,B 0,C 180,E1 -6317.318,E2 -6317.318} C_VEL
LIN {X 0,Y 495.769,Z 220.216,A -85,B 0,C 180,E1 -6319.89,E2 -6319.89} C_VEL
LIN {X 0,Y 495.756,Z 220.229,A -85,B 0,C 180,E1 -6322.86,E2 -6322.86} C_VEL
LIN {X 0,Y 495.778,Z 220.227,A -85,B 0,C 180,E1 -6326.068,E2 -6326.068} C_VEL
LIN {X 0,Y 495.769,Z 220.225,A -85,B 0,C 180,E1 -6328.814,E2 -6328.814} C_VEL
LIN {X 0,Y 495.753,Z 220.231,A -85,B 0,C 180,E1 -6331.725,E2 -6331.725} C_VEL
LIN {X 0,Y 495.771,Z 220.221,A -85,B 0,C 180,E1 -6334.695,E2 -6334.695} C_VEL
LIN {X 0,Y 495.728,Z 220.233,A -85,B 0,C 180,E1 -6337.561,E2 -6337.561} C_VEL
LIN {X 0,Y 495.764,Z 220.222,A -85,B 0,C 180,E1 -6340.699,E2 -6340.699} C_VEL
LIN {X 0,Y 495.731,Z 220.236,A -85,B 0,C 180,E1 -6343.695,E2 -6343.695} C_VEL
LIN {X 0,Y 495.725,Z 220.222,A -85,B 0,C 180,E1 -6346.305,E2 -6346.305} C_VEL
LIN {X 0,Y 495.776,Z 220.215,A -85,B 0,C 180,E1 -6349.301,E2 -6349.301} C_VEL
LIN {X 0,Y 495.728,Z 220.232,A -85,B 0,C 180,E1 -6352.438,E2 -6352.438} C_VEL
LIN {X 0,Y 495.779,Z 220.218,A -85,B 0,C 180,E1 -6355.457,E2 -6355.457} C_VEL
LIN {X 0,Y 495.755,Z 220.229,A -85,B 0,C 180,E1 -6358.364,E2 -6358.364} C_VEL
LIN {X 0,Y 495.749,Z 220.22,A -85,B 0,C 180,E1 -6360.757,E2 -6360.757} C_VEL
LIN {X 0,Y 495.092,Z 220.309,A -85,B 0,C 180,E1 -6361.436,E2 -6361.436} C_VEL
LIN {X 0,Y 492.236,Z 220.667,A -85,B 0,C 180,E1 -6362.539,E2 -6362.539} C_VEL
LIN {X 0,Y 489.827,Z 220.973,A -85,B 0,C 180,E1 -6363.428,E2 -6363.428} C_VEL
LIN {X 0,Y 488.811,Z 221.095,A -85,B 0,C 180,E1 -6364.114,E2 -6364.114} C_VEL
LIN {X 0,Y 488.739,Z 221.103,A -85,B 0,C 180,E1 -6364.346,E2 -6364.346} C_VEL
LIN {X 0,Y 488.719,Z 221.11,A -85,B 0,C 180,E1 -6367.153,E2 -6367.153} C_VEL
LIN {X 0,Y 488.725,Z 221.108,A -85,B 0,C 180,E1 -6369.811,E2 -6369.811} C_VEL
LIN {X 0,Y 488.731,Z 221.105,A -85,B 0,C 180,E1 -6372.423,E2 -6372.423} C_VEL
LIN {X 0,Y 488.761,Z 221.105,A -85,B 0,C 180,E1 -6375,E2 -6375} C_VEL
LIN {X 0,Y 488.802,Z 221.097,A -85,B 0,C 180,E1 -6378.388,E2 -6378.388} C_VEL
LIN {X 0,Y 488.815,Z 221.097,A -85,B 0,C 180,E1 -6381.734,E2 -6381.734} C_VEL
LIN {X 0,Y 488.856,Z 221.09,A -85,B 0,C 180,E1 -6384.224,E2 -6384.224} C_VEL
LIN {X 0,Y 488.959,Z 221.079,A -85,B 0,C 180,E1 -6387.529,E2 -6387.529} C_VEL
LIN {X 0,Y 488.951,Z 221.082,A -85,B 0,C 180,E1 -6390.824,E2 -6390.824} C_VEL
LIN {X 0,Y 488.959,Z 221.079,A -85,B 0,C 180,E1 -6392.471,E2 -6392.471} C_VEL
LIN {X 0,Y 488.856,Z 221.09,A -85,B 0,C 180,E1 -6395.776,E2 -6395.776} C_VEL
LIN {X 0,Y 488.815,Z 221.097,A -85,B 0,C 180,E1 -6398.266,E2 -6398.266} C_VEL
LIN {X 0,Y 488.802,Z 221.097,A -85,B 0,C 180,E1 -6401.612,E2 -6401.612} C_VEL
LIN {X 0,Y 488.761,Z 221.105,A -85,B 0,C 180,E1 -6405,E2 -6405} C_VEL
LIN {X 0,Y 488.751,Z 221.107,A -85,B 0,C 180,E1 -6408.442,E2 -6408.442} C_VEL
LIN {X 0,Y 488.703,Z 221.11,A -85,B 0,C 180,E1 -6411.071,E2 -6411.071} C_VEL
LIN {X 0,Y 488.685,Z 221.11,A -85,B 0,C 180,E1 -6413.746,E2 -6413.746} C_VEL
LIN {X 0,Y 488.788,Z 221.099,A -85,B 0,C 180,E1 -6416.944,E2 -6416.944} C_VEL
LIN {X 0,Y 488.706,Z 221.105,A -85,B 0,C 180,E1 -6420.363,E2 -6420.363} C_VEL
LIN {X 0,Y 488.732,Z 221.099,A -85,B 0,C 180,E1 -6423.485,E2 -6423.485} C_VEL
LIN {X 0,Y 488.684,Z 221.11,A -85,B 0,C 180,E1 -6426.356,E2 -6426.356} C_VEL
LIN {X 0,Y 488.739,Z 221.1,A -85,B 0,C 180,E1 -6429.25,E2 -6429.25} C_VEL
LIN {X 0,Y 488.708,Z 221.093,A -85,B 0,C 180,E1 -6431.601,E2 -6431.601} C_VEL
LIN {X 0,Y 488.709,Z 221.104,A -85,B 0,C 180,E1 -6434.802,E2 -6434.802} C_VEL
LIN {X 0,Y 488.727,Z 221.105,A -85,B 0,C 180,E1 -6437.479,E2 -6437.479} C_VEL
LIN {X 0,Y 488.737,Z 221.101,A -85,B 0,C 180,E1 -6440.75,E2 -6440.75} C_VEL
LIN {X 0,Y 488.681,Z 221.113,A -85,B 0,C 180,E1 -6443.869,E2 -6443.869} C_VEL
LIN {X 0,Y 488.736,Z 221.099,A -85,B 0,C 180,E1 -6446.878,E2 -6446.878} C_VEL
LIN {X 0,Y 488.721,Z 221.11,A -85,B 0,C 180,E1 -6449.781,E2 -6449.781} C_VEL
LIN {X 0,Y 488.789,Z 221.085,A -85,B 0,C 180,E1 -6453.057,E2 -6453.057} C_VEL
LIN {X 0,Y 488.674,Z 221.111,A -85,B 0,C 180,E1 -6456.254,E2 -6456.254} C_VEL
LIN {X 0,Y 488.744,Z 221.101,A -85,B 0,C 180,E1 -6459.176,E2 -6459.176} C_VEL
LIN {X 0,Y 488.732,Z 221.097,A -85,B 0,C 180,E1 -6462.424,E2 -6462.424} C_VEL
LIN {X 0,Y 488.763,Z 221.1,A -85,B 0,C 180,E1 -6465,E2 -6465} C_VEL
LIN {X 0,Y 488.804,Z 221.087,A -85,B 0,C 180,E1 -6468.388,E2 -6468.388} C_VEL
LIN {X 0,Y 488.817,Z 221.091,A -85,B 0,C 180,E1 -6471.734,E2 -6471.734} C_VEL
LIN {X 0,Y 488.847,Z 221.088,A -85,B 0,C 180,E1 -6474.225,E2 -6474.225} C_VEL
LIN {X 0,Y 488.961,Z 221.071,A -85,B 0,C 180,E1 -6477.529,E2 -6477.529} C_VEL
LIN {X 0,Y 488.933,Z 221.067,A -85,B 0,C 180,E1 -6480.824,E2 -6480.824} C_VEL
LIN {X 0,Y 488.961,Z 221.07,A -85,B 0,C 180,E1 -6482.472,E2 -6482.472} C_VEL
LIN {X 0,Y 488.842,Z 221.088,A -85,B 0,C 180,E1 -6485.776,E2 -6485.776} C_VEL
LIN {X 0,Y 488.785,Z 221.089,A -85,B 0,C 180,E1 -6488.267,E2 -6488.267} C_VEL
LIN {X 0,Y 488.805,Z 221.09,A -85,B 0,C 180,E1 -6491.613,E2 -6491.613} C_VEL
LIN {X 0,Y 488.762,Z 221.103,A -85,B 0,C 180,E1 -6495.001,E2 -6495.001} C_VEL
LIN {X 0,Y 488.747,Z 221.093,A -85,B 0,C 180,E1 -6498.443,E2 -6498.443} C_VEL
LIN {X 0,Y 488.707,Z 221.108,A -85,B 0,C 180,E1 -6501.071,E2 -6501.071} C_VEL
LIN {X 0,Y 488.689,Z 221.106,A -85,B 0,C 180,E1 -6503.746,E2 -6503.746} C_VEL
LIN {X 0,Y 488.792,Z 221.091,A -85,B 0,C 180,E1 -6506.944,E2 -6506.944} C_VEL
LIN {X 0,Y 488.709,Z 221.11,A -85,B 0,C 180,E1 -6510.363,E2 -6510.363} C_VEL
LIN {X 0,Y 488.711,Z 221.098,A -85,B 0,C 180,E1 -6513.48,E2 -6513.48} C_VEL
LIN {X 0,Y 488.683,Z 221.112,A -85,B 0,C 180,E1 -6516.355,E2 -6516.355} C_VEL
LIN {X 0,Y 488.701,Z 221.102,A -85,B 0,C 180,E1 -6519.255,E2 -6519.255} C_VEL
LIN {X 0,Y 488.708,Z 221.105,A -85,B 0,C 180,E1 -6521.6,E2 -6521.6} C_VEL
LIN {X 0,Y 488.703,Z 221.107,A -85,B 0,C 180,E1 -6524.803,E2 -6524.803} C_VEL
LIN {X 0,Y 488.693,Z 221.108,A -85,B 0,C 180,E1 -6527.475,E2 -6527.475} C_VEL
LIN {X 0,Y 488.735,Z 221.095,A -85,B 0,C 180,E1 -6529.677,E2 -6529.677} C_VEL
LIN {X 0,Y 488.681,Z 221.109,A -85,B 0,C 180,E1 -6532.841,E2 -6532.841} C_VEL
LIN {X 0,Y 488.732,Z 221.107,A -85,B 0,C 180,E1 -6535.888,E2 -6535.888} C_VEL
LIN {X 0,Y 488.694,Z 221.111,A -85,B 0,C 180,E1 -6538.821,E2 -6538.821} C_VEL
LIN {X 0,Y 488.716,Z 221.109,A -85,B 0,C 180,E1 -6541.67,E2 -6541.67} C_VEL
LIN {X 0,Y 488.79,Z 221.308,A -85,B 0,C 180,E1 -6543.111,E2 -6543.111} C_VEL
LIN {X 0,Y 490.233,Z 229.586,A -85,B 0,C 180,E1 -6545.045,E2 -6545.045} C_VEL
LIN {X 0,Y 490.096,Z 236.677,A -85,B 0,C 180,E1 -6546.602,E2 -6546.602} C_VEL
LIN {X 0,Y 489.545,Z 252.008,A -85,B 0,C 180,E1 -6549.846,E2 -6549.846} C_VEL
LIN {X 0,Y 489.07,Z 265.435,A -85,B 0,C 180,E1 -6552.652,E2 -6552.652} C_VEL
LIN {X 0,Y 488.967,Z 270.561,A -85,B 0,C 180,E1 -6553.713,E2 -6553.713} C_VEL
LIN {X 0,Y 490.584,Z 280.175,A -85,B 0,C 180,E1 -6553.941,E2 -6553.941} C_VEL
LIN {X 0,Y 491.654,Z 287.085,A -85,B 0,C 180,E1 -6554.08,E2 -6554.08} C_VEL
LIN {X 0,Y 491.131,Z 375.366,A -85,B 0,C 180,E1 -6555.392,E2 -6555.392} C_VEL
LIN {X 0,Y 490.905,Z 386.138,A -85,B 0,C 180,E1 -6555.65,E2 -6555.65} C_VEL
LIN {X 0,Y 490.643,Z 395.24,A -85,B 0,C 180,E1 -6555.959,E2 -6555.959} C_VEL
LIN {X 0,Y 490.364,Z 405.607,A -85,B 0,C 180,E1 -6556.427,E2 -6556.427} C_VEL
LIN {X 0,Y 490.051,Z 414.747,A -85,B 0,C 180,E1 -6556.946,E2 -6556.946} C_VEL
LIN {X 0,Y 489.694,Z 423.742,A -85,B 0,C 180,E1 -6557.568,E2 -6557.568} C_VEL
LIN {X 0,Y 489.404,Z 432.475,A -85,B 0,C 180,E1 -6558.297,E2 -6558.297} C_VEL
LIN {X 0,Y 489.062,Z 439.871,A -85,B 0,C 180,E1 -6559.024,E2 -6559.024} C_VEL
LIN {X 0,Y 488.783,Z 447.092,A -85,B 0,C 180,E1 -6559.855,E2 -6559.855} C_VEL
LIN {X 0,Y 488.549,Z 453.295,A -85,B 0,C 180,E1 -6560.687,E2 -6560.687} C_VEL
LIN {X 0,Y 488.32,Z 459.832,A -85,B 0,C 180,E1 -6561.725,E2 -6561.725} C_VEL
LIN {X 0,Y 488.187,Z 464.333,A -85,B 0,C 180,E1 -6562.556,E2 -6562.556} C_VEL
LIN {X 0,Y 488.017,Z 469.823,A -85,B 0,C 180,E1 -6563.8,E2 -6563.8} C_VEL
LIN {X 0,Y 487.968,Z 474.144,A -85,B 0,C 180,E1 -6565.043,E2 -6565.043} C_VEL
LIN {X 0,Y 487.929,Z 476.507,A -85,B 0,C 180,E1 -6565.87,E2 -6565.87} C_VEL
LIN {X 0,Y 487.965,Z 478.304,A -85,B 0,C 180,E1 -6566.697,E2 -6566.697} C_VEL
LIN {X 0,Y 487.891,Z 480.743,A -85,B 0,C 180,E1 -6568.349,E2 -6568.349} C_VEL
LIN {X 0,Y 487.835,Z 481.329,A -85,B 0,C 180,E1 -6569.175,E2 -6569.175} C_VEL
LIN {X 0,Y 487.835,Z 481.329,A -85,B 0,C 180,E1 -6570.825,E2 -6570.825} C_VEL
LIN {X 0,Y 487.891,Z 480.743,A -85,B 0,C 180,E1 -6571.651,E2 -6571.651} C_VEL
LIN {X 0,Y 487.965,Z 478.304,A -85,B 0,C 180,E1 -6573.303,E2 -6573.303} C_VEL
LIN {X 0,Y 487.923,Z 475.358,A -85,B 0,C 180,E1 -6574.544,E2 -6574.544} C_VEL
LIN {X 0,Y 488.012,Z 471.375,A -85,B 0,C 180,E1 -6575.786,E2 -6575.786} C_VEL
LIN {X 0,Y 488.044,Z 468.162,A -85,B 0,C 180,E1 -6576.615,E2 -6576.615} C_VEL
LIN {X 0,Y 488.227,Z 462.142,A -85,B 0,C 180,E1 -6577.86,E2 -6577.86} C_VEL
LIN {X 0,Y 488.449,Z 456.047,A -85,B 0,C 180,E1 -6578.898,E2 -6578.898} C_VEL
LIN {X 0,Y 488.675,Z 450.346,A -85,B 0,C 180,E1 -6579.729,E2 -6579.729} C_VEL
LIN {X 0,Y 488.964,Z 441.79,A -85,B 0,C 180,E1 -6580.769,E2 -6580.769} C_VEL
LIN {X 0,Y 489.321,Z 433.609,A -85,B 0,C 180,E1 -6581.6,E2 -6581.6} C_VEL
LIN {X 0,Y 489.644,Z 425.095,A -85,B 0,C 180,E1 -6582.328,E2 -6582.328} C_VEL
LIN {X 0,Y 489.951,Z 416.81,A -85,B 0,C 180,E1 -6582.924,E2 -6582.924} C_VEL
LIN {X 0,Y 490.334,Z 406.614,A -85,B 0,C 180,E1 -6583.521,E2 -6583.521} C_VEL
LIN {X 0,Y 490.63,Z 396.529,A -85,B 0,C 180,E1 -6583.988,E2 -6583.988} C_VEL
LIN {X 0,Y 490.9,Z 387.013,A -85,B 0,C 180,E1 -6584.324,E2 -6584.324} C_VEL
LIN {X 0,Y 491.154,Z 376.699,A -85,B 0,C 180,E1 -6584.581,E2 -6584.581} C_VEL
LIN {X 0,Y 491.592,Z 300.033,A -85,B 0,C 180,E1 -6585.73,E2 -6585.73} C_VEL
LIN {X 0,Y 491.464,Z 285.601,A -85,B 0,C 180,E1 -6585.949,E2 -6585.949} C_VEL
LIN {X 0,Y 488.949,Z 270.69,A -85,B 0,C 180,E1 -6586.278,E2 -6586.278} C_VEL
LIN {X 0,Y 488.933,Z 269.875,A -85,B 0,C 180,E1 -6586.385,E2 -6586.385} C_VEL
LIN {X 0,Y 489.353,Z 257.315,A -85,B 0,C 180,E1 -6589.077,E2 -6589.077} C_VEL
LIN {X 0,Y 489.814,Z 244.799,A -85,B 0,C 180,E1 -6591.683,E2 -6591.683} C_VEL
LIN {X 0,Y 490.34,Z 231.345,A -85,B 0,C 180,E1 -6594.56,E2 -6594.56} C_VEL
LIN {X 0,Y 489.335,Z 224.168,A -85,B 0,C 180,E1 -6596.209,E2 -6596.209} C_VEL
LIN {X 0,Y 488.789,Z 221.126,A -85,B 0,C 180,E1 -6596.962,E2 -6596.962} C_VEL
LIN {X 0,Y 488.712,Z 221.111,A -85,B 0,C 180,E1 -6600.363,E2 -6600.363} C_VEL
LIN {X 0,Y 488.737,Z 221.105,A -85,B 0,C 180,E1 -6603.484,E2 -6603.484} C_VEL
LIN {X 0,Y 488.684,Z 221.11,A -85,B 0,C 180,E1 -6606.354,E2 -6606.354} C_VEL
LIN {X 0,Y 488.703,Z 221.107,A -85,B 0,C 180,E1 -6609.254,E2 -6609.254} C_VEL
LIN {X 0,Y 488.708,Z 221.102,A -85,B 0,C 180,E1 -6611.599,E2 -6611.599} C_VEL
LIN {X 0,Y 488.703,Z 221.105,A -85,B 0,C 180,E1 -6614.802,E2 -6614.802} C_VEL
LIN {X 0,Y 488.693,Z 221.113,A -85,B 0,C 180,E1 -6617.474,E2 -6617.474} C_VEL
LIN {X 0,Y 488.734,Z 221.103,A -85,B 0,C 180,E1 -6619.676,E2 -6619.676} C_VEL
LIN {X 0,Y 488.68,Z 221.11,A -85,B 0,C 180,E1 -6622.841,E2 -6622.841} C_VEL
LIN {X 0,Y 488.721,Z 221.1,A -85,B 0,C 180,E1 -6625.886,E2 -6625.886} C_VEL
LIN {X 0,Y 488.691,Z 221.108,A -85,B 0,C 180,E1 -6628.82,E2 -6628.82} C_VEL
LIN {X 0,Y 488.744,Z 221.098,A -85,B 0,C 180,E1 -6631.671,E2 -6631.671} C_VEL
LIN {X 0,Y 488.74,Z 221.095,A -85,B 0,C 180,E1 -6634.443,E2 -6634.443} C_VEL
LIN {X 0,Y 488.723,Z 221.109,A -85,B 0,C 180,E1 -6637.153,E2 -6637.153} C_VEL
LIN {X 0,Y 488.725,Z 221.096,A -85,B 0,C 180,E1 -6639.81,E2 -6639.81} C_VEL
LIN {X 0,Y 488.714,Z 221.095,A -85,B 0,C 180,E1 -6642.422,E2 -6642.422} C_VEL
LIN {X 0,Y 488.762,Z 221.103,A -85,B 0,C 180,E1 -6644.999,E2 -6644.999} C_VEL
LIN {X 0,Y 488.805,Z 221.09,A -85,B 0,C 180,E1 -6648.387,E2 -6648.387} C_VEL
LIN {X 0,Y 488.785,Z 221.089,A -85,B 0,C 180,E1 -6651.733,E2 -6651.733} C_VEL
LIN {X 0,Y 488.842,Z 221.088,A -85,B 0,C 180,E1 -6654.224,E2 -6654.224} C_VEL
LIN {X 0,Y 488.961,Z 221.07,A -85,B 0,C 180,E1 -6657.528,E2 -6657.528} C_VEL
LIN {X 0,Y 488.934,Z 221.07,A -85,B 0,C 180,E1 -6660.823,E2 -6660.823} C_VEL
LIN {X 0,Y 488.961,Z 221.071,A -85,B 0,C 180,E1 -6662.471,E2 -6662.471} C_VEL
LIN {X 0,Y 488.847,Z 221.088,A -85,B 0,C 180,E1 -6665.775,E2 -6665.775} C_VEL
LIN {X 0,Y 488.817,Z 221.091,A -85,B 0,C 180,E1 -6668.266,E2 -6668.266} C_VEL
LIN {X 0,Y 488.804,Z 221.087,A -85,B 0,C 180,E1 -6671.612,E2 -6671.612} C_VEL
LIN {X 0,Y 488.763,Z 221.1,A -85,B 0,C 180,E1 -6675,E2 -6675} C_VEL
LIN {X 0,Y 488.753,Z 221.094,A -85,B 0,C 180,E1 -6678.442,E2 -6678.442} C_VEL
LIN {X 0,Y 488.704,Z 221.103,A -85,B 0,C 180,E1 -6681.07,E2 -6681.07} C_VEL
LIN {X 0,Y 488.677,Z 221.111,A -85,B 0,C 180,E1 -6683.746,E2 -6683.746} C_VEL
LIN {X 0,Y 488.789,Z 221.085,A -85,B 0,C 180,E1 -6686.943,E2 -6686.943} C_VEL
LIN {X 0,Y 488.707,Z 221.112,A -85,B 0,C 180,E1 -6690.363,E2 -6690.363} C_VEL
LIN {X 0,Y 488.732,Z 221.1,A -85,B 0,C 180,E1 -6693.484,E2 -6693.484} C_VEL
LIN {X 0,Y 488.684,Z 221.113,A -85,B 0,C 180,E1 -6696.355,E2 -6696.355} C_VEL
LIN {X 0,Y 488.698,Z 221.106,A -85,B 0,C 180,E1 -6699.254,E2 -6699.254} C_VEL
LIN {X 0,Y 488.727,Z 221.105,A -85,B 0,C 180,E1 -6702.521,E2 -6702.521} C_VEL
LIN {X 0,Y 488.709,Z 221.104,A -85,B 0,C 180,E1 -6705.198,E2 -6705.198} C_VEL
LIN {X 0,Y 488.708,Z 221.093,A -85,B 0,C 180,E1 -6708.399,E2 -6708.399} C_VEL
LIN {X 0,Y 488.737,Z 221.101,A -85,B 0,C 180,E1 -6710.942,E2 -6710.942} C_VEL
LIN {X 0,Y 488.68,Z 221.107,A -85,B 0,C 180,E1 -6713.868,E2 -6713.868} C_VEL
LIN {X 0,Y 488.735,Z 221.099,A -85,B 0,C 180,E1 -6716.877,E2 -6716.877} C_VEL
LIN {X 0,Y 488.72,Z 221.101,A -85,B 0,C 180,E1 -6719.781,E2 -6719.781} C_VEL
LIN {X 0,Y 488.788,Z 221.099,A -85,B 0,C 180,E1 -6723.056,E2 -6723.056} C_VEL
LIN {X 0,Y 488.739,Z 221.103,A -85,B 0,C 180,E1 -6724.346,E2 -6724.346} C_VEL
LIN {X 0,Y 488.094,Z 221.187,A -85,B 0,C 180,E1 -6725.034,E2 -6725.034} C_VEL
LIN {X 0,Y 485.226,Z 221.546,A -85,B 0,C 180,E1 -6726.151,E2 -6726.151} C_VEL
LIN {X 0,Y 482.779,Z 221.852,A -85,B 0,C 180,E1 -6727.05,E2 -6727.05} C_VEL
LIN {X 0,Y 481.721,Z 221.982,A -85,B 0,C 180,E1 -6727.746,E2 -6727.746} C_VEL
LIN {X 0,Y 481.632,Z 221.991,A -85,B 0,C 180,E1 -6727.981,E2 -6727.981} C_VEL
LIN {X 0,Y 481.704,Z 221.98,A -85,B 0,C 180,E1 -6730.393,E2 -6730.393} C_VEL
LIN {X 0,Y 481.688,Z 221.986,A -85,B 0,C 180,E1 -6733.034,E2 -6733.034} C_VEL
LIN {X 0,Y 481.691,Z 221.986,A -85,B 0,C 180,E1 -6735.639,E2 -6735.639} C_VEL
LIN {X 0,Y 481.748,Z 221.976,A -85,B 0,C 180,E1 -6738.215,E2 -6738.215} C_VEL
LIN {X 0,Y 481.76,Z 221.977,A -85,B 0,C 180,E1 -6741.612,E2 -6741.612} C_VEL
LIN {X 0,Y 481.816,Z 221.967,A -85,B 0,C 180,E1 -6744.14,E2 -6744.14} C_VEL
LIN {X 0,Y 481.926,Z 221.956,A -85,B 0,C 180,E1 -6747.493,E2 -6747.493} C_VEL
LIN {X 0,Y 481.902,Z 221.96,A -85,B 0,C 180,E1 -6750.836,E2 -6750.836} C_VEL
LIN {X 0,Y 481.926,Z 221.956,A -85,B 0,C 180,E1 -6752.507,E2 -6752.507} C_VEL
LIN {X 0,Y 481.816,Z 221.967,A -85,B 0,C 180,E1 -6755.86,E2 -6755.86} C_VEL
LIN {X 0,Y 481.76,Z 221.977,A -85,B 0,C 180,E1 -6758.388,E2 -6758.388} C_VEL
LIN {X 0,Y 481.748,Z 221.975,A -85,B 0,C 180,E1 -6761.785,E2 -6761.785} C_VEL
LIN {X 0,Y 481.741,Z 221.978,A -85,B 0,C 180,E1 -6765.224,E2 -6765.224} C_VEL
LIN {X 0,Y 481.709,Z 221.985,A -85,B 0,C 180,E1 -6768.722,E2 -6768.722} C_VEL
LIN {X 0,Y 481.642,Z 221.988,A -85,B 0,C 180,E1 -6771.395,E2 -6771.395} C_VEL
LIN {X 0,Y 481.67,Z 221.987,A -85,B 0,C 180,E1 -6774.113,E2 -6774.113} C_VEL
LIN {X 0,Y 481.743,Z 221.975,A -85,B 0,C 180,E1 -6777.139,E2 -6777.139} C_VEL
LIN {X 0,Y 481.675,Z 221.972,A -85,B 0,C 180,E1 -6779.741,E2 -6779.741} C_VEL
LIN {X 0,Y 481.67,Z 221.983,A -85,B 0,C 180,E1 -6782.674,E2 -6782.674} C_VEL
LIN {X 0,Y 481.638,Z 221.979,A -85,B 0,C 180,E1 -6785.709,E2 -6785.709} C_VEL
LIN {X 0,Y 481.711,Z 221.976,A -85,B 0,C 180,E1 -6789.354,E2 -6789.354} C_VEL
LIN {X 0,Y 481.645,Z 221.97,A -85,B 0,C 180,E1 -6792.161,E2 -6792.161} C_VEL
LIN {X 0,Y 481.657,Z 221.983,A -85,B 0,C 180,E1 -6795.543,E2 -6795.543} C_VEL
LIN {X 0,Y 481.669,Z 221.984,A -85,B 0,C 180,E1 -6798.085,E2 -6798.085} C_VEL
LIN {X 0,Y 481.693,Z 221.979,A -85,B 0,C 180,E1 -6801.144,E2 -6801.144} C_VEL
LIN {X 0,Y 481.664,Z 221.977,A -85,B 0,C 180,E1 -6804.795,E2 -6804.795} C_VEL
LIN {X 0,Y 481.669,Z 221.981,A -85,B 0,C 180,E1 -6807.326,E2 -6807.326} C_VEL
LIN {X 0,Y 481.676,Z 221.981,A -85,B 0,C 180,E1 -6810.259,E2 -6810.259} C_VEL
LIN {X 0,Y 481.742,Z 221.963,A -85,B 0,C 180,E1 -6813.112,E2 -6813.112} C_VEL
LIN {X 0,Y 481.656,Z 221.989,A -85,B 0,C 180,E1 -6815.886,E2 -6815.886} C_VEL
LIN {X 0,Y 481.7,Z 221.977,A -85,B 0,C 180,E1 -6819.028,E2 -6819.028} C_VEL
LIN {X 0,Y 481.705,Z 221.973,A -85,B 0,C 180,E1 -6822.159,E2 -6822.159} C_VEL
LIN {X 0,Y 481.742,Z 221.973,A -85,B 0,C 180,E1 -6824.776,E2 -6824.776} C_VEL
LIN {X 0,Y 481.749,Z 221.966,A -85,B 0,C 180,E1 -6828.216,E2 -6828.216} C_VEL
LIN {X 0,Y 481.762,Z 221.97,A -85,B 0,C 180,E1 -6831.612,E2 -6831.612} C_VEL
LIN {X 0,Y 481.808,Z 221.965,A -85,B 0,C 180,E1 -6834.14,E2 -6834.14} C_VEL
LIN {X 0,Y 481.927,Z 221.947,A -85,B 0,C 180,E1 -6837.493,E2 -6837.493} C_VEL
LIN {X 0,Y 481.885,Z 221.945,A -85,B 0,C 180,E1 -6840.836,E2 -6840.836} C_VEL
LIN {X 0,Y 481.928,Z 221.946,A -85,B 0,C 180,E1 -6842.508,E2 -6842.508} C_VEL
LIN {X 0,Y 481.8,Z 221.965,A -85,B 0,C 180,E1 -6845.861,E2 -6845.861} C_VEL
LIN {X 0,Y 481.739,Z 221.966,A -85,B 0,C 180,E1 -6848.389,E2 -6848.389} C_VEL
LIN {X 0,Y 481.751,Z 221.967,A -85,B 0,C 180,E1 -6851.785,E2 -6851.785} C_VEL
LIN {X 0,Y 481.742,Z 221.974,A -85,B 0,C 180,E1 -6855.225,E2 -6855.225} C_VEL
LIN {X 0,Y 481.708,Z 221.969,A -85,B 0,C 180,E1 -6858.722,E2 -6858.722} C_VEL
LIN {X 0,Y 481.646,Z 221.984,A -85,B 0,C 180,E1 -6861.395,E2 -6861.395} C_VEL
LIN {X 0,Y 481.674,Z 221.982,A -85,B 0,C 180,E1 -6864.114,E2 -6864.114} C_VEL
LIN {X 0,Y 481.747,Z 221.967,A -85,B 0,C 180,E1 -6867.139,E2 -6867.139} C_VEL
LIN {X 0,Y 481.679,Z 221.98,A -85,B 0,C 180,E1 -6869.742,E2 -6869.742} C_VEL
LIN {X 0,Y 481.653,Z 221.984,A -85,B 0,C 180,E1 -6872.676,E2 -6872.676} C_VEL
LIN {X 0,Y 481.636,Z 221.984,A -85,B 0,C 180,E1 -6875.71,E2 -6875.71} C_VEL
LIN {X 0,Y 481.671,Z 221.981,A -85,B 0,C 180,E1 -6878.86,E2 -6878.86} C_VEL
LIN {X 0,Y 481.654,Z 221.986,A -85,B 0,C 180,E1 -6881.913,E2 -6881.913} C_VEL
LIN {X 0,Y 481.656,Z 221.987,A -85,B 0,C 180,E1 -6884.458,E2 -6884.458} C_VEL
LIN {X 0,Y 481.649,Z 221.988,A -85,B 0,C 180,E1 -6887.84,E2 -6887.84} C_VEL
LIN {X 0,Y 481.682,Z 221.982,A -85,B 0,C 180,E1 -6890.652,E2 -6890.652} C_VEL
LIN {X 0,Y 481.629,Z 221.987,A -85,B 0,C 180,E1 -6893.377,E2 -6893.377} C_VEL
LIN {X 0,Y 481.712,Z 221.981,A -85,B 0,C 180,E1 -6896.33,E2 -6896.33} C_VEL
LIN {X 0,Y 481.653,Z 221.99,A -85,B 0,C 180,E1 -6899.418,E2 -6899.418} C_VEL
LIN {X 0,Y 481.73,Z 222.012,A -85,B 0,C 180,E1 -6902.836,E2 -6902.836} C_VEL
LIN {X 0,Y 483.288,Z 231.207,A -85,B 0,C 180,E1 -6905.057,E2 -6905.057} C_VEL
LIN {X 0,Y 483.034,Z 239.42,A -85,B 0,C 180,E1 -6906.869,E2 -6906.869} C_VEL
LIN {X 0,Y 482.531,Z 253.91,A -85,B 0,C 180,E1 -6909.985,E2 -6909.985} C_VEL
LIN {X 0,Y 481.985,Z 268.241,A -85,B 0,C 180,E1 -6913.045,E2 -6913.045} C_VEL
LIN {X 0,Y 481.97,Z 270.376,A -85,B 0,C 180,E1 -6913.47,E2 -6913.47} C_VEL
LIN {X 0,Y 483.437,Z 279.136,A -85,B 0,C 180,E1 -6913.685,E2 -6913.685} C_VEL
LIN {X 0,Y 484.816,Z 288.308,A -85,B 0,C 180,E1 -6913.87,E2 -6913.87} C_VEL
LIN {X 0,Y 484.269,Z 375.174,A -85,B 0,C 180,E1 -6915.18,E2 -6915.18} C_VEL
LIN {X 0,Y 484.047,Z 385.945,A -85,B 0,C 180,E1 -6915.442,E2 -6915.442} C_VEL
LIN {X 0,Y 483.764,Z 395.048,A -85,B 0,C 180,E1 -6915.755,E2 -6915.755} C_VEL
LIN {X 0,Y 483.454,Z 405.414,A -85,B 0,C 180,E1 -6916.229,E2 -6916.229} C_VEL
LIN {X 0,Y 483.125,Z 414.554,A -85,B 0,C 180,E1 -6916.755,E2 -6916.755} C_VEL
LIN {X 0,Y 482.713,Z 423.548,A -85,B 0,C 180,E1 -6917.386,E2 -6917.386} C_VEL
LIN {X 0,Y 482.434,Z 432.288,A -85,B 0,C 180,E1 -6918.126,E2 -6918.126} C_VEL
LIN {X 0,Y 482.06,Z 439.677,A -85,B 0,C 180,E1 -6918.862,E2 -6918.862} C_VEL
LIN {X 0,Y 481.739,Z 446.897,A -85,B 0,C 180,E1 -6919.705,E2 -6919.705} C_VEL
LIN {X 0,Y 481.496,Z 453.1,A -85,B 0,C 180,E1 -6920.549,E2 -6920.549} C_VEL
LIN {X 0,Y 481.268,Z 459.638,A -85,B 0,C 180,E1 -6921.603,E2 -6921.603} C_VEL
LIN {X 0,Y 481.103,Z 464.139,A -85,B 0,C 180,E1 -6922.445,E2 -6922.445} C_VEL
LIN {X 0,Y 480.917,Z 470.092,A -85,B 0,C 180,E1 -6923.834,E2 -6923.834} C_VEL
LIN {X 0,Y 480.898,Z 473.951,A -85,B 0,C 180,E1 -6924.97,E2 -6924.97} C_VEL
LIN {X 0,Y 480.829,Z 476.314,A -85,B 0,C 180,E1 -6925.809,E2 -6925.809} C_VEL
LIN {X 0,Y 480.889,Z 478.112,A -85,B 0,C 180,E1 -6926.649,E2 -6926.649} C_VEL
LIN {X 0,Y 480.793,Z 480.55,A -85,B 0,C 180,E1 -6928.325,E2 -6928.325} C_VEL
LIN {X 0,Y 480.761,Z 481.137,A -85,B 0,C 180,E1 -6929.162,E2 -6929.162} C_VEL
LIN {X 0,Y 480.761,Z 481.137,A -85,B 0,C 180,E1 -6930.838,E2 -6930.838} C_VEL
LIN {X 0,Y 480.793,Z 480.55,A -85,B 0,C 180,E1 -6931.675,E2 -6931.675} C_VEL
LIN {X 0,Y 480.889,Z 478.112,A -85,B 0,C 180,E1 -6933.351,E2 -6933.351} C_VEL
LIN {X 0,Y 480.841,Z 475.165,A -85,B 0,C 180,E1 -6934.611,E2 -6934.611} C_VEL
LIN {X 0,Y 480.918,Z 471.181,A -85,B 0,C 180,E1 -6935.871,E2 -6935.871} C_VEL
LIN {X 0,Y 481.021,Z 466.054,A -85,B 0,C 180,E1 -6937.134,E2 -6937.134} C_VEL
LIN {X 0,Y 481.226,Z 460.794,A -85,B 0,C 180,E1 -6938.186,E2 -6938.186} C_VEL
LIN {X 0,Y 481.45,Z 454.477,A -85,B 0,C 180,E1 -6939.24,E2 -6939.24} C_VEL
LIN {X 0,Y 481.671,Z 448.525,A -85,B 0,C 180,E1 -6940.084,E2 -6940.084} C_VEL
LIN {X 0,Y 481.982,Z 441.597,A -85,B 0,C 180,E1 -6940.927,E2 -6940.927} C_VEL
LIN {X 0,Y 482.346,Z 433.416,A -85,B 0,C 180,E1 -6941.77,E2 -6941.77} C_VEL
LIN {X 0,Y 482.644,Z 426.254,A -85,B 0,C 180,E1 -6942.403,E2 -6942.403} C_VEL
LIN {X 0,Y 483.037,Z 416.187,A -85,B 0,C 180,E1 -6943.14,E2 -6943.14} C_VEL
LIN {X 0,Y 483.412,Z 406.421,A -85,B 0,C 180,E1 -6943.719,E2 -6943.719} C_VEL
LIN {X 0,Y 483.725,Z 396.336,A -85,B 0,C 180,E1 -6944.192,E2 -6944.192} C_VEL
LIN {X 0,Y 484.037,Z 386.82,A -85,B 0,C 180,E1 -6944.532,E2 -6944.532} C_VEL
LIN {X 0,Y 484.301,Z 376.507,A -85,B 0,C 180,E1 -6944.792,E2 -6944.792} C_VEL
LIN {X 0,Y 484.704,Z 301.945,A -85,B 0,C 180,E1 -6945.928,E2 -6945.928} C_VEL
LIN {X 0,Y 484.678,Z 286.619,A -85,B 0,C 180,E1 -6946.16,E2 -6946.16} C_VEL
LIN {X 0,Y 481.94,Z 270.574,A -85,B 0,C 180,E1 -6946.517,E2 -6946.517} C_VEL
LIN {X 0,Y 481.935,Z 269.683,A -85,B 0,C 180,E1 -6946.63,E2 -6946.63} C_VEL
LIN {X 0,Y 482.481,Z 256.17,A -85,B 0,C 180,E1 -6949.574,E2 -6949.574} C_VEL
LIN {X 0,Y 482.981,Z 241.522,A -85,B 0,C 180,E1 -6952.681,E2 -6952.681} C_VEL
LIN {X 0,Y 483.323,Z 231.208,A -85,B 0,C 180,E1 -6954.941,E2 -6954.941} C_VEL
LIN {X 0,Y 481.73,Z 222.005,A -85,B 0,C 180,E1 -6957.164,E2 -6957.164} C_VEL
LIN {X 0,Y 481.653,Z 221.99,A -85,B 0,C 180,E1 -6960.582,E2 -6960.582} C_VEL
LIN {X 0,Y 481.699,Z 221.984,A -85,B 0,C 180,E1 -6963.733,E2 -6963.733} C_VEL
LIN {X 0,Y 481.628,Z 221.987,A -85,B 0,C 180,E1 -6966.747,E2 -6966.747} C_VEL
LIN {X 0,Y 481.679,Z 221.975,A -85,B 0,C 180,E1 -6969.94,E2 -6969.94} C_VEL
LIN {X 0,Y 481.64,Z 221.988,A -85,B 0,C 180,E1 -6973.3,E2 -6973.3} C_VEL
LIN {X 0,Y 481.655,Z 221.987,A -85,B 0,C 180,E1 -6975.641,E2 -6975.641} C_VEL
LIN {X 0,Y 481.657,Z 221.984,A -85,B 0,C 180,E1 -6978.958,E2 -6978.958} C_VEL
LIN {X 0,Y 481.655,Z 221.987,A -85,B 0,C 180,E1 -6981.992,E2 -6981.992} C_VEL
LIN {X 0,Y 481.684,Z 221.98,A -85,B 0,C 180,E1 -6985.317,E2 -6985.317} C_VEL
LIN {X 0,Y 481.643,Z 221.985,A -85,B 0,C 180,E1 -6988.311,E2 -6988.311} C_VEL
LIN {X 0,Y 481.7,Z 221.982,A -85,B 0,C 180,E1 -6991.218,E2 -6991.218} C_VEL
LIN {X 0,Y 481.698,Z 221.973,A -85,B 0,C 180,E1 -6994.042,E2 -6994.042} C_VEL
LIN {X 0,Y 481.675,Z 221.983,A -85,B 0,C 180,E1 -6996.811,E2 -6996.811} C_VEL
LIN {X 0,Y 481.695,Z 221.975,A -85,B 0,C 180,E1 -6999.502,E2 -6999.502} C_VEL
LIN {X 0,Y 481.691,Z 221.968,A -85,B 0,C 180,E1 -7002.157,E2 -7002.157} C_VEL
LIN {X 0,Y 481.742,Z 221.974,A -85,B 0,C 180,E1 -7004.775,E2 -7004.775} C_VEL
LIN {X 0,Y 481.751,Z 221.967,A -85,B 0,C 180,E1 -7008.215,E2 -7008.215} C_VEL
LIN {X 0,Y 481.739,Z 221.966,A -85,B 0,C 180,E1 -7011.611,E2 -7011.611} C_VEL
LIN {X 0,Y 481.8,Z 221.965,A -85,B 0,C 180,E1 -7014.139,E2 -7014.139} C_VEL
LIN {X 0,Y 481.928,Z 221.946,A -85,B 0,C 180,E1 -7017.492,E2 -7017.492} C_VEL
LIN {X 0,Y 481.885,Z 221.947,A -85,B 0,C 180,E1 -7020.835,E2 -7020.835} C_VEL
LIN {X 0,Y 481.927,Z 221.947,A -85,B 0,C 180,E1 -7022.507,E2 -7022.507} C_VEL
LIN {X 0,Y 481.808,Z 221.965,A -85,B 0,C 180,E1 -7025.86,E2 -7025.86} C_VEL
LIN {X 0,Y 481.762,Z 221.97,A -85,B 0,C 180,E1 -7028.388,E2 -7028.388} C_VEL
LIN {X 0,Y 481.749,Z 221.966,A -85,B 0,C 180,E1 -7031.784,E2 -7031.784} C_VEL
LIN {X 0,Y 481.742,Z 221.973,A -85,B 0,C 180,E1 -7035.224,E2 -7035.224} C_VEL
LIN {X 0,Y 481.71,Z 221.968,A -85,B 0,C 180,E1 -7038.721,E2 -7038.721} C_VEL
LIN {X 0,Y 481.643,Z 221.982,A -85,B 0,C 180,E1 -7041.394,E2 -7041.394} C_VEL
LIN {X 0,Y 481.658,Z 221.989,A -85,B 0,C 180,E1 -7044.114,E2 -7044.114} C_VEL
LIN {X 0,Y 481.744,Z 221.961,A -85,B 0,C 180,E1 -7047.139,E2 -7047.139} C_VEL
LIN {X 0,Y 481.676,Z 221.981,A -85,B 0,C 180,E1 -7049.741,E2 -7049.741} C_VEL
LIN {X 0,Y 481.669,Z 221.981,A -85,B 0,C 180,E1 -7052.674,E2 -7052.674} C_VEL
LIN {X 0,Y 481.638,Z 221.983,A -85,B 0,C 180,E1 -7055.709,E2 -7055.709} C_VEL
LIN {X 0,Y 481.668,Z 221.982,A -85,B 0,C 180,E1 -7058.859,E2 -7058.859} C_VEL
LIN {X 0,Y 481.669,Z 221.988,A -85,B 0,C 180,E1 -7062.158,E2 -7062.158} C_VEL
LIN {X 0,Y 481.657,Z 221.983,A -85,B 0,C 180,E1 -7064.457,E2 -7064.457} C_VEL
LIN {X 0,Y 481.645,Z 221.97,A -85,B 0,C 180,E1 -7067.839,E2 -7067.839} C_VEL
LIN {X 0,Y 481.711,Z 221.976,A -85,B 0,C 180,E1 -7070.646,E2 -7070.646} C_VEL
LIN {X 0,Y 481.638,Z 221.979,A -85,B 0,C 180,E1 -7074.291,E2 -7074.291} C_VEL
LIN {X 0,Y 481.67,Z 221.983,A -85,B 0,C 180,E1 -7077.326,E2 -7077.326} C_VEL
LIN {X 0,Y 481.675,Z 221.973,A -85,B 0,C 180,E1 -7080.259,E2 -7080.259} C_VEL
LIN {X 0,Y 481.742,Z 221.977,A -85,B 0,C 180,E1 -7083.112,E2 -7083.112} C_VEL
LIN {X 0,Y 481.67,Z 221.987,A -85,B 0,C 180,E1 -7085.887,E2 -7085.887} C_VEL
LIN {X 0,Y 481.632,Z 221.991,A -85,B 0,C 180,E1 -7087.981,E2 -7087.981} C_VEL
LIN {X 0,Y 480.964,Z 222.073,A -85,B 0,C 180,E1 -7088.679,E2 -7088.679} C_VEL
LIN {X 0,Y 478.138,Z 222.427,A -85,B 0,C 180,E1 -7089.814,E2 -7089.814} C_VEL
LIN {X 0,Y 475.754,Z 222.726,A -85,B 0,C 180,E1 -7090.728,E2 -7090.728} C_VEL
LIN {X 0,Y 474.734,Z 222.854,A -85,B 0,C 180,E1 -7091.434,E2 -7091.434} C_VEL
LIN {X 0,Y 474.652,Z 222.862,A -85,B 0,C 180,E1 -7091.673,E2 -7091.673} C_VEL
LIN {X 0,Y 474.697,Z 222.854,A -85,B 0,C 180,E1 -7094.544,E2 -7094.544} C_VEL
LIN {X 0,Y 474.701,Z 222.854,A -85,B 0,C 180,E1 -7098.038,E2 -7098.038} C_VEL
LIN {X 0,Y 474.725,Z 222.854,A -85,B 0,C 180,E1 -7101.486,E2 -7101.486} C_VEL
LIN {X 0,Y 474.779,Z 222.844,A -85,B 0,C 180,E1 -7104.052,E2 -7104.052} C_VEL
LIN {X 0,Y 474.892,Z 222.833,A -85,B 0,C 180,E1 -7107.455,E2 -7107.455} C_VEL
LIN {X 0,Y 474.909,Z 222.828,A -85,B 0,C 180,E1 -7110,E2 -7110} C_VEL
LIN {X 0,Y 474.892,Z 222.832,A -85,B 0,C 180,E1 -7112.545,E2 -7112.545} C_VEL
LIN {X 0,Y 474.779,Z 222.844,A -85,B 0,C 180,E1 -7115.948,E2 -7115.948} C_VEL
LIN {X 0,Y 474.725,Z 222.854,A -85,B 0,C 180,E1 -7118.514,E2 -7118.514} C_VEL
LIN {X 0,Y 474.701,Z 222.854,A -85,B 0,C 180,E1 -7121.962,E2 -7121.962} C_VEL
LIN {X 0,Y 474.697,Z 222.854,A -85,B 0,C 180,E1 -7125.456,E2 -7125.456} C_VEL
LIN {X 0,Y 474.662,Z 222.861,A -85,B 0,C 180,E1 -7129.01,E2 -7129.01} C_VEL
LIN {X 0,Y 474.585,Z 222.867,A -85,B 0,C 180,E1 -7131.729,E2 -7131.729} C_VEL
LIN {X 0,Y 474.653,Z 222.863,A -85,B 0,C 180,E1 -7134.493,E2 -7134.493} C_VEL
LIN {X 0,Y 474.695,Z 222.853,A -85,B 0,C 180,E1 -7137.339,E2 -7137.339} C_VEL
LIN {X 0,Y 474.602,Z 222.866,A -85,B 0,C 180,E1 -7140.811,E2 -7140.811} C_VEL
LIN {X 0,Y 474.634,Z 222.853,A -85,B 0,C 180,E1 -7143.984,E2 -7143.984} C_VEL
LIN {X 0,Y 474.571,Z 222.868,A -85,B 0,C 180,E1 -7146.9,E2 -7146.9} C_VEL
LIN {X 0,Y 474.647,Z 222.858,A -85,B 0,C 180,E1 -7149.651,E2 -7149.651} C_VEL
LIN {X 0,Y 474.611,Z 222.848,A -85,B 0,C 180,E1 -7152.934,E2 -7152.934} C_VEL
LIN {X 0,Y 474.615,Z 222.864,A -85,B 0,C 180,E1 -7155.897,E2 -7155.897} C_VEL
LIN {X 0,Y 474.641,Z 222.852,A -85,B 0,C 180,E1 -7159.039,E2 -7159.039} C_VEL
LIN {X 0,Y 474.613,Z 222.865,A -85,B 0,C 180,E1 -7161.703,E2 -7161.703} C_VEL
LIN {X 0,Y 474.625,Z 222.854,A -85,B 0,C 180,E1 -7164.726,E2 -7164.726} C_VEL
LIN {X 0,Y 474.633,Z 222.863,A -85,B 0,C 180,E1 -7167.788,E2 -7167.788} C_VEL
LIN {X 0,Y 474.621,Z 222.858,A -85,B 0,C 180,E1 -7170.885,E2 -7170.885} C_VEL
LIN {X 0,Y 474.651,Z 222.851,A -85,B 0,C 180,E1 -7173.628,E2 -7173.628} C_VEL
LIN {X 0,Y 474.632,Z 222.859,A -85,B 0,C 180,E1 -7176.642,E2 -7176.642} C_VEL
LIN {X 0,Y 474.652,Z 222.845,A -85,B 0,C 180,E1 -7180.09,E2 -7180.09} C_VEL
LIN {X 0,Y 474.649,Z 222.851,A -85,B 0,C 180,E1 -7182.775,E2 -7182.775} C_VEL
LIN {X 0,Y 474.65,Z 222.863,A -85,B 0,C 180,E1 -7185.422,E2 -7185.422} C_VEL
LIN {X 0,Y 474.703,Z 222.844,A -85,B 0,C 180,E1 -7188.038,E2 -7188.038} C_VEL
LIN {X 0,Y 474.727,Z 222.843,A -85,B 0,C 180,E1 -7191.487,E2 -7191.487} C_VEL
LIN {X 0,Y 474.77,Z 222.842,A -85,B 0,C 180,E1 -7194.053,E2 -7194.053} C_VEL
LIN {X 0,Y 474.893,Z 222.823,A -85,B 0,C 180,E1 -7197.456,E2 -7197.456} C_VEL
LIN {X 0,Y 474.911,Z 222.809,A -85,B 0,C 180,E1 -7200,E2 -7200} C_VEL
LIN {X 0,Y 474.894,Z 222.823,A -85,B 0,C 180,E1 -7202.545,E2 -7202.545} C_VEL
LIN {X 0,Y 474.761,Z 222.841,A -85,B 0,C 180,E1 -7205.948,E2 -7205.948} C_VEL
LIN {X 0,Y 474.711,Z 222.843,A -85,B 0,C 180,E1 -7208.514,E2 -7208.514} C_VEL
LIN {X 0,Y 474.704,Z 222.845,A -85,B 0,C 180,E1 -7211.963,E2 -7211.963} C_VEL
LIN {X 0,Y 474.7,Z 222.849,A -85,B 0,C 180,E1 -7215.456,E2 -7215.456} C_VEL
LIN {X 0,Y 474.663,Z 222.847,A -85,B 0,C 180,E1 -7219.011,E2 -7219.011} C_VEL
LIN {X 0,Y 474.588,Z 222.862,A -85,B 0,C 180,E1 -7221.729,E2 -7221.729} C_VEL
LIN {X 0,Y 474.656,Z 222.86,A -85,B 0,C 180,E1 -7224.493,E2 -7224.493} C_VEL
LIN {X 0,Y 474.681,Z 222.845,A -85,B 0,C 180,E1 -7227.335,E2 -7227.335} C_VEL
LIN {X 0,Y 474.605,Z 222.865,A -85,B 0,C 180,E1 -7230.231,E2 -7230.231} C_VEL
LIN {X 0,Y 474.615,Z 222.855,A -85,B 0,C 180,E1 -7233.223,E2 -7233.223} C_VEL
LIN {X 0,Y 474.589,Z 222.867,A -85,B 0,C 180,E1 -7236.324,E2 -7236.324} C_VEL
LIN {X 0,Y 474.619,Z 222.857,A -85,B 0,C 180,E1 -7239.647,E2 -7239.647} C_VEL
LIN {X 0,Y 474.616,Z 222.862,A -85,B 0,C 180,E1 -7242.935,E2 -7242.935} C_VEL
LIN {X 0,Y 474.608,Z 222.864,A -85,B 0,C 180,E1 -7245.895,E2 -7245.895} C_VEL
LIN {X 0,Y 474.629,Z 222.85,A -85,B 0,C 180,E1 -7249.041,E2 -7249.041} C_VEL
LIN {X 0,Y 474.612,Z 222.863,A -85,B 0,C 180,E1 -7251.704,E2 -7251.704} C_VEL
LIN {X 0,Y 474.626,Z 222.859,A -85,B 0,C 180,E1 -7254.726,E2 -7254.726} C_VEL
LIN {X 0,Y 474.638,Z 222.859,A -85,B 0,C 180,E1 -7257.788,E2 -7257.788} C_VEL
LIN {X 0,Y 474.609,Z 222.867,A -85,B 0,C 180,E1 -7260.889,E2 -7260.889} C_VEL
LIN {X 0,Y 474.68,Z 222.976,A -85,B 0,C 180,E1 -7262.679,E2 -7262.679} C_VEL
LIN {X 0,Y 476.275,Z 232.091,A -85,B 0,C 180,E1 -7264.898,E2 -7264.898} C_VEL
LIN {X 0,Y 476.22,Z 237.846,A -85,B 0,C 180,E1 -7266.205,E2 -7266.205} C_VEL
LIN {X 0,Y 475.6,Z 252.709,A -85,B 0,C 180,E1 -7269.454,E2 -7269.454} C_VEL
LIN {X 0,Y 475.057,Z 266.107,A -85,B 0,C 180,E1 -7272.346,E2 -7272.346} C_VEL
LIN {X 0,Y 474.951,Z 270.065,A -85,B 0,C 180,E1 -7273.204,E2 -7273.204} C_VEL
LIN {X 0,Y 475.605,Z 274.279,A -85,B 0,C 180,E1 -7273.337,E2 -7273.337} C_VEL
LIN {X 0,Y 478.007,Z 288.576,A -85,B 0,C 180,E1 -7273.641,E2 -7273.641} C_VEL
LIN {X 0,Y 477.423,Z 374.981,A -85,B 0,C 180,E1 -7274.963,E2 -7274.963} C_VEL
LIN {X 0,Y 477.176,Z 385.753,A -85,B 0,C 180,E1 -7275.227,E2 -7275.227} C_VEL
LIN {X 0,Y 476.892,Z 394.855,A -85,B 0,C 180,E1 -7275.546,E2 -7275.546} C_VEL
LIN {X 0,Y 476.607,Z 404.214,A -85,B 0,C 180,E1 -7275.973,E2 -7275.973} C_VEL
LIN {X 0,Y 476.198,Z 414.36,A -85,B 0,C 180,E1 -7276.559,E2 -7276.559} C_VEL
LIN {X 0,Y 475.766,Z 423.355,A -85,B 0,C 180,E1 -7277.198,E2 -7277.198} C_VEL
LIN {X 0,Y 475.457,Z 432.19,A -85,B 0,C 180,E1 -7277.958,E2 -7277.958} C_VEL
LIN {X 0,Y 475.071,Z 439.483,A -85,B 0,C 180,E1 -7278.696,E2 -7278.696} C_VEL
LIN {X 0,Y 474.726,Z 446.704,A -85,B 0,C 180,E1 -7279.551,E2 -7279.551} C_VEL
LIN {X 0,Y 474.467,Z 452.907,A -85,B 0,C 180,E1 -7280.408,E2 -7280.408} C_VEL
LIN {X 0,Y 474.201,Z 459.445,A -85,B 0,C 180,E1 -7281.477,E2 -7281.477} C_VEL
LIN {X 0,Y 474.033,Z 463.946,A -85,B 0,C 180,E1 -7282.332,E2 -7282.332} C_VEL
LIN {X 0,Y 473.868,Z 469.244,A -85,B 0,C 180,E1 -7283.561,E2 -7283.561} C_VEL
LIN {X 0,Y 473.828,Z 473.758,A -85,B 0,C 180,E1 -7284.894,E2 -7284.894} C_VEL
LIN {X 0,Y 473.736,Z 476.121,A -85,B 0,C 180,E1 -7285.746,E2 -7285.746} C_VEL
LIN {X 0,Y 473.796,Z 477.919,A -85,B 0,C 180,E1 -7286.598,E2 -7286.598} C_VEL
LIN {X 0,Y 473.698,Z 480.358,A -85,B 0,C 180,E1 -7288.3,E2 -7288.3} C_VEL
LIN {X 0,Y 473.689,Z 480.945,A -85,B 0,C 180,E1 -7289.15,E2 -7289.15} C_VEL
LIN {X 0,Y 473.689,Z 480.945,A -85,B 0,C 180,E1 -7290.85,E2 -7290.85} C_VEL
LIN {X 0,Y 473.698,Z 480.358,A -85,B 0,C 180,E1 -7291.7,E2 -7291.7} C_VEL
LIN {X 0,Y 473.796,Z 477.919,A -85,B 0,C 180,E1 -7293.402,E2 -7293.402} C_VEL
LIN {X 0,Y 473.764,Z 474.973,A -85,B 0,C 180,E1 -7294.68,E2 -7294.68} C_VEL
LIN {X 0,Y 473.826,Z 470.988,A -85,B 0,C 180,E1 -7295.96,E2 -7295.96} C_VEL
LIN {X 0,Y 473.947,Z 465.86,A -85,B 0,C 180,E1 -7297.241,E2 -7297.241} C_VEL
LIN {X 0,Y 474.162,Z 460.6,A -85,B 0,C 180,E1 -7298.309,E2 -7298.309} C_VEL
LIN {X 0,Y 474.399,Z 454.283,A -85,B 0,C 180,E1 -7299.379,E2 -7299.379} C_VEL
LIN {X 0,Y 474.634,Z 448.331,A -85,B 0,C 180,E1 -7300.235,E2 -7300.235} C_VEL
LIN {X 0,Y 474.973,Z 441.403,A -85,B 0,C 180,E1 -7301.09,E2 -7301.09} C_VEL
LIN {X 0,Y 475.374,Z 433.222,A -85,B 0,C 180,E1 -7301.945,E2 -7301.945} C_VEL
LIN {X 0,Y 475.684,Z 425.301,A -85,B 0,C 180,E1 -7302.648,E2 -7302.648} C_VEL
LIN {X 0,Y 476.106,Z 415.994,A -85,B 0,C 180,E1 -7303.335,E2 -7303.335} C_VEL
LIN {X 0,Y 476.504,Z 406.228,A -85,B 0,C 180,E1 -7303.922,E2 -7303.922} C_VEL
LIN {X 0,Y 476.846,Z 396.143,A -85,B 0,C 180,E1 -7304.401,E2 -7304.401} C_VEL
LIN {X 0,Y 477.17,Z 386.627,A -85,B 0,C 180,E1 -7304.745,E2 -7304.745} C_VEL
LIN {X 0,Y 477.451,Z 376.315,A -85,B 0,C 180,E1 -7305.009,E2 -7305.009} C_VEL
LIN {X 0,Y 477.888,Z 306.166,A -85,B 0,C 180,E1 -7306.093,E2 -7306.093} C_VEL
LIN {X 0,Y 477.951,Z 288.072,A -85,B 0,C 180,E1 -7306.368,E2 -7306.368} C_VEL
LIN {X 0,Y 474.954,Z 270.386,A -85,B 0,C 180,E1 -7306.767,E2 -7306.767} C_VEL
LIN {X 0,Y 474.929,Z 269.492,A -85,B 0,C 180,E1 -7306.883,E2 -7306.883} C_VEL
LIN {X 0,Y 475.475,Z 257.038,A -85,B 0,C 180,E1 -7309.65,E2 -7309.65} C_VEL
LIN {X 0,Y 476.034,Z 242.435,A -85,B 0,C 180,E1 -7312.802,E2 -7312.802} C_VEL
LIN {X 0,Y 476.402,Z 233.115,A -85,B 0,C 180,E1 -7314.862,E2 -7314.862} C_VEL
LIN {X 0,Y 474.89,Z 223.9,A -85,B 0,C 180,E1 -7317.07,E2 -7317.07} C_VEL
LIN {X 0,Y 474.669,Z 222.871,A -85,B 0,C 180,E1 -7317.418,E2 -7317.418} C_VEL
LIN {X 0,Y 474.607,Z 222.867,A -85,B 0,C 180,E1 -7320.81,E2 -7320.81} C_VEL
LIN {X 0,Y 474.64,Z 222.865,A -85,B 0,C 180,E1 -7323.983,E2 -7323.983} C_VEL
LIN {X 0,Y 474.574,Z 222.866,A -85,B 0,C 180,E1 -7326.899,E2 -7326.899} C_VEL
LIN {X 0,Y 474.629,Z 222.856,A -85,B 0,C 180,E1 -7329.647,E2 -7329.647} C_VEL
LIN {X 0,Y 474.616,Z 222.861,A -85,B 0,C 180,E1 -7332.934,E2 -7332.934} C_VEL
LIN {X 0,Y 474.608,Z 222.866,A -85,B 0,C 180,E1 -7335.894,E2 -7335.894} C_VEL
LIN {X 0,Y 474.629,Z 222.86,A -85,B 0,C 180,E1 -7339.04,E2 -7339.04} C_VEL
LIN {X 0,Y 474.611,Z 222.868,A -85,B 0,C 180,E1 -7341.704,E2 -7341.704} C_VEL
LIN {X 0,Y 474.623,Z 222.857,A -85,B 0,C 180,E1 -7344.725,E2 -7344.725} C_VEL
LIN {X 0,Y 474.628,Z 222.863,A -85,B 0,C 180,E1 -7347.787,E2 -7347.787} C_VEL
LIN {X 0,Y 474.624,Z 222.861,A -85,B 0,C 180,E1 -7350.884,E2 -7350.884} C_VEL
LIN {X 0,Y 474.659,Z 222.852,A -85,B 0,C 180,E1 -7353.628,E2 -7353.628} C_VEL
LIN {X 0,Y 474.636,Z 222.858,A -85,B 0,C 180,E1 -7356.641,E2 -7356.641} C_VEL
LIN {X 0,Y 474.654,Z 222.847,A -85,B 0,C 180,E1 -7360.089,E2 -7360.089} C_VEL
LIN {X 0,Y 474.638,Z 222.85,A -85,B 0,C 180,E1 -7362.774,E2 -7362.774} C_VEL
LIN {X 0,Y 474.648,Z 222.859,A -85,B 0,C 180,E1 -7365.421,E2 -7365.421} C_VEL
LIN {X 0,Y 474.704,Z 222.845,A -85,B 0,C 180,E1 -7368.037,E2 -7368.037} C_VEL
LIN {X 0,Y 474.711,Z 222.843,A -85,B 0,C 180,E1 -7371.486,E2 -7371.486} C_VEL
LIN {X 0,Y 474.748,Z 222.851,A -85,B 0,C 180,E1 -7374.904,E2 -7374.904} C_VEL
LIN {X 0,Y 474.894,Z 222.823,A -85,B 0,C 180,E1 -7377.455,E2 -7377.455} C_VEL
LIN {X 0,Y 474.911,Z 222.809,A -85,B 0,C 180,E1 -7380,E2 -7380} C_VEL
LIN {X 0,Y 474.893,Z 222.823,A -85,B 0,C 180,E1 -7382.544,E2 -7382.544} C_VEL
LIN {X 0,Y 474.77,Z 222.842,A -85,B 0,C 180,E1 -7385.947,E2 -7385.947} C_VEL
LIN {X 0,Y 474.727,Z 222.843,A -85,B 0,C 180,E1 -7388.513,E2 -7388.513} C_VEL
LIN {X 0,Y 474.703,Z 222.844,A -85,B 0,C 180,E1 -7391.962,E2 -7391.962} C_VEL
LIN {X 0,Y 474.699,Z 222.85,A -85,B 0,C 180,E1 -7395.455,E2 -7395.455} C_VEL
LIN {X 0,Y 474.663,Z 222.843,A -85,B 0,C 180,E1 -7399.01,E2 -7399.01} C_VEL
LIN {X 0,Y 474.586,Z 222.862,A -85,B 0,C 180,E1 -7401.728,E2 -7401.728} C_VEL
LIN {X 0,Y 474.638,Z 222.861,A -85,B 0,C 180,E1 -7404.493,E2 -7404.493} C_VEL
LIN {X 0,Y 474.678,Z 222.841,A -85,B 0,C 180,E1 -7407.334,E2 -7407.334} C_VEL
LIN {X 0,Y 474.603,Z 222.869,A -85,B 0,C 180,E1 -7410.23,E2 -7410.23} C_VEL
LIN {X 0,Y 474.64,Z 222.855,A -85,B 0,C 180,E1 -7413.22,E2 -7413.22} C_VEL
LIN {X 0,Y 474.589,Z 222.869,A -85,B 0,C 180,E1 -7416.323,E2 -7416.323} C_VEL
LIN {X 0,Y 474.625,Z 222.862,A -85,B 0,C 180,E1 -7419.647,E2 -7419.647} C_VEL
LIN {X 0,Y 474.648,Z 222.857,A -85,B 0,C 180,E1 -7422.93,E2 -7422.93} C_VEL
LIN {X 0,Y 474.606,Z 222.857,A -85,B 0,C 180,E1 -7425.895,E2 -7425.895} C_VEL
LIN {X 0,Y 474.637,Z 222.844,A -85,B 0,C 180,E1 -7429.039,E2 -7429.039} C_VEL
LIN {X 0,Y 474.613,Z 222.868,A -85,B 0,C 180,E1 -7431.703,E2 -7431.703} C_VEL
LIN {X 0,Y 474.625,Z 222.85,A -85,B 0,C 180,E1 -7434.726,E2 -7434.726} C_VEL
LIN {X 0,Y 474.634,Z 222.866,A -85,B 0,C 180,E1 -7437.788,E2 -7437.788} C_VEL
LIN {X 0,Y 474.62,Z 222.852,A -85,B 0,C 180,E1 -7440.884,E2 -7440.884} C_VEL
LIN {X 0,Y 474.657,Z 222.863,A -85,B 0,C 180,E1 -7443.628,E2 -7443.628} C_VEL
LIN {X 0,Y 474.632,Z 222.861,A -85,B 0,C 180,E1 -7446.641,E2 -7446.641} C_VEL
LIN {X 0,Y 474.653,Z 222.859,A -85,B 0,C 180,E1 -7450.09,E2 -7450.09} C_VEL
LIN {X 0,Y 474.652,Z 222.862,A -85,B 0,C 180,E1 -7451.673,E2 -7451.673} C_VEL
LIN {X 0,Y 473.989,Z 222.943,A -85,B 0,C 180,E1 -7452.382,E2 -7452.382} C_VEL
LIN {X 0,Y 471.14,Z 223.302,A -85,B 0,C 180,E1 -7453.533,E2 -7453.533} C_VEL
LIN {X 0,Y 468.725,Z 223.604,A -85,B 0,C 180,E1 -7454.462,E2 -7454.462} C_VEL
LIN {X 0,Y 467.683,Z 223.731,A -85,B 0,C 180,E1 -7455.179,E2 -7455.179} C_VEL
LIN {X 0,Y 467.596,Z 223.74,A -85,B 0,C 180,E1 -7455.422,E2 -7455.422} C_VEL
LIN {X 0,Y 467.65,Z 223.734,A -85,B 0,C 180,E1 -7458.734,E2 -7458.734} C_VEL
LIN {X 0,Y 467.745,Z 223.721,A -85,B 0,C 180,E1 -7462.228,E2 -7462.228} C_VEL
LIN {X 0,Y 467.723,Z 223.726,A -85,B 0,C 180,E1 -7464.827,E2 -7464.827} C_VEL
LIN {X 0,Y 467.857,Z 223.709,A -85,B 0,C 180,E1 -7467.417,E2 -7467.417} C_VEL
LIN {X 0,Y 467.88,Z 223.704,A -85,B 0,C 180,E1 -7470,E2 -7470} C_VEL
LIN {X 0,Y 467.857,Z 223.709,A -85,B 0,C 180,E1 -7472.583,E2 -7472.583} C_VEL
LIN {X 0,Y 467.743,Z 223.721,A -85,B 0,C 180,E1 -7476.037,E2 -7476.037} C_VEL
LIN {X 0,Y 467.679,Z 223.732,A -85,B 0,C 180,E1 -7478.643,E2 -7478.643} C_VEL
LIN {X 0,Y 467.652,Z 223.733,A -85,B 0,C 180,E1 -7482.145,E2 -7482.145} C_VEL
LIN {X 0,Y 467.636,Z 223.734,A -85,B 0,C 180,E1 -7485.695,E2 -7485.695} C_VEL
LIN {X 0,Y 467.614,Z 223.74,A -85,B 0,C 180,E1 -7488.765,E2 -7488.765} C_VEL
LIN {X 0,Y 467.576,Z 223.741,A -85,B 0,C 180,E1 -7491.268,E2 -7491.268} C_VEL
LIN {X 0,Y 467.568,Z 223.743,A -85,B 0,C 180,E1 -7493.943,E2 -7493.943} C_VEL
LIN {X 0,Y 467.613,Z 223.739,A -85,B 0,C 180,E1 -7496.8,E2 -7496.8} C_VEL
LIN {X 0,Y 467.55,Z 223.731,A -85,B 0,C 180,E1 -7499.738,E2 -7499.738} C_VEL
LIN {X 0,Y 467.58,Z 223.737,A -85,B 0,C 180,E1 -7502.758,E2 -7502.758} C_VEL
LIN {X 0,Y 467.552,Z 223.734,A -85,B 0,C 180,E1 -7505.89,E2 -7505.89} C_VEL
LIN {X 0,Y 467.596,Z 223.734,A -85,B 0,C 180,E1 -7509.143,E2 -7509.143} C_VEL
LIN {X 0,Y 467.583,Z 223.721,A -85,B 0,C 180,E1 -7512.567,E2 -7512.567} C_VEL
LIN {X 0,Y 467.567,Z 223.736,A -85,B 0,C 180,E1 -7515.053,E2 -7515.053} C_VEL
LIN {X 0,Y 467.606,Z 223.736,A -85,B 0,C 180,E1 -7517.443,E2 -7517.443} C_VEL
LIN {X 0,Y 467.596,Z 223.735,A -85,B 0,C 180,E1 -7520.857,E2 -7520.857} C_VEL
LIN {X 0,Y 467.559,Z 223.737,A -85,B 0,C 180,E1 -7524.261,E2 -7524.261} C_VEL
LIN {X 0,Y 467.579,Z 223.736,A -85,B 0,C 180,E1 -7527.321,E2 -7527.321} C_VEL
LIN {X 0,Y 467.567,Z 223.736,A -85,B 0,C 180,E1 -7530.668,E2 -7530.668} C_VEL
LIN {X 0,Y 467.61,Z 223.723,A -85,B 0,C 180,E1 -7533.2,E2 -7533.2} C_VEL
LIN {X 0,Y 467.587,Z 223.737,A -85,B 0,C 180,E1 -7536.469,E2 -7536.469} C_VEL
LIN {X 0,Y 467.62,Z 223.724,A -85,B 0,C 180,E1 -7539.778,E2 -7539.778} C_VEL
LIN {X 0,Y 467.607,Z 223.728,A -85,B 0,C 180,E1 -7542.507,E2 -7542.507} C_VEL
LIN {X 0,Y 467.608,Z 223.738,A -85,B 0,C 180,E1 -7545.197,E2 -7545.197} C_VEL
LIN {X 0,Y 467.654,Z 223.723,A -85,B 0,C 180,E1 -7547.855,E2 -7547.855} C_VEL
LIN {X 0,Y 467.68,Z 223.717,A -85,B 0,C 180,E1 -7551.358,E2 -7551.358} C_VEL
LIN {X 0,Y 467.734,Z 223.719,A -85,B 0,C 180,E1 -7553.963,E2 -7553.963} C_VEL
LIN {X 0,Y 467.858,Z 223.699,A -85,B 0,C 180,E1 -7557.418,E2 -7557.418} C_VEL
LIN {X 0,Y 467.881,Z 223.684,A -85,B 0,C 180,E1 -7560,E2 -7560} C_VEL
LIN {X 0,Y 467.859,Z 223.699,A -85,B 0,C 180,E1 -7562.583,E2 -7562.583} C_VEL
LIN {X 0,Y 467.723,Z 223.718,A -85,B 0,C 180,E1 -7566.038,E2 -7566.038} C_VEL
LIN {X 0,Y 467.669,Z 223.72,A -85,B 0,C 180,E1 -7568.643,E2 -7568.643} C_VEL
LIN {X 0,Y 467.656,Z 223.723,A -85,B 0,C 180,E1 -7572.146,E2 -7572.146} C_VEL
LIN {X 0,Y 467.639,Z 223.727,A -85,B 0,C 180,E1 -7575.695,E2 -7575.695} C_VEL
LIN {X 0,Y 467.622,Z 223.725,A -85,B 0,C 180,E1 -7579.308,E2 -7579.308} C_VEL
LIN {X 0,Y 467.535,Z 223.742,A -85,B 0,C 180,E1 -7582.074,E2 -7582.074} C_VEL
LIN {X 0,Y 467.595,Z 223.734,A -85,B 0,C 180,E1 -7584.888,E2 -7584.888} C_VEL
LIN {X 0,Y 467.62,Z 223.724,A -85,B 0,C 180,E1 -7587.769,E2 -7587.769} C_VEL
LIN {X 0,Y 467.568,Z 223.741,A -85,B 0,C 180,E1 -7591.045,E2 -7591.045} C_VEL
LIN {X 0,Y 467.577,Z 223.733,A -85,B 0,C 180,E1 -7594.24,E2 -7594.24} C_VEL
LIN {X 0,Y 467.548,Z 223.742,A -85,B 0,C 180,E1 -7597.187,E2 -7597.187} C_VEL
LIN {X 0,Y 467.576,Z 223.737,A -85,B 0,C 180,E1 -7600.265,E2 -7600.265} C_VEL
LIN {X 0,Y 467.588,Z 223.741,A -85,B 0,C 180,E1 -7602.567,E2 -7602.567} C_VEL
LIN {X 0,Y 467.567,Z 223.739,A -85,B 0,C 180,E1 -7605.053,E2 -7605.053} C_VEL
LIN {X 0,Y 467.591,Z 223.737,A -85,B 0,C 180,E1 -7607.44,E2 -7607.44} C_VEL
LIN {X 0,Y 467.584,Z 223.737,A -85,B 0,C 180,E1 -7610.856,E2 -7610.856} C_VEL
LIN {X 0,Y 467.562,Z 223.737,A -85,B 0,C 180,E1 -7614.261,E2 -7614.261} C_VEL
LIN {X 0,Y 467.584,Z 223.737,A -85,B 0,C 180,E1 -7617.321,E2 -7617.321} C_VEL
LIN {X 0,Y 467.559,Z 223.744,A -85,B 0,C 180,E1 -7620.671,E2 -7620.671} C_VEL
LIN {X 0,Y 467.654,Z 223.966,A -85,B 0,C 180,E1 -7622.51,E2 -7622.51} C_VEL
LIN {X 0,Y 469.276,Z 232.975,A -85,B 0,C 180,E1 -7624.734,E2 -7624.734} C_VEL
LIN {X 0,Y 469.275,Z 238.432,A -85,B 0,C 180,E1 -7626.002,E2 -7626.002} C_VEL
LIN {X 0,Y 468.611,Z 253.576,A -85,B 0,C 180,E1 -7629.363,E2 -7629.363} C_VEL
LIN {X 0,Y 468.084,Z 265.92,A -85,B 0,C 180,E1 -7632.074,E2 -7632.074} C_VEL
LIN {X 0,Y 467.913,Z 269.85,A -85,B 0,C 180,E1 -7632.941,E2 -7632.941} C_VEL
LIN {X 0,Y 468.43,Z 273.022,A -85,B 0,C 180,E1 -7633.058,E2 -7633.058} C_VEL
LIN {X 0,Y 471.199,Z 289.464,A -85,B 0,C 180,E1 -7633.415,E2 -7633.415} C_VEL
LIN {X 0,Y 470.582,Z 374.789,A -85,B 0,C 180,E1 -7634.739,E2 -7634.739} C_VEL
LIN {X 0,Y 470.332,Z 384.685,A -85,B 0,C 180,E1 -7634.98,E2 -7634.98} C_VEL
LIN {X 0,Y 470.024,Z 394.663,A -85,B 0,C 180,E1 -7635.33,E2 -7635.33} C_VEL
LIN {X 0,Y 469.712,Z 404.021,A -85,B 0,C 180,E1 -7635.762,E2 -7635.762} C_VEL
LIN {X 0,Y 469.27,Z 414.164,A -85,B 0,C 180,E1 -7636.357,E2 -7636.357} C_VEL
LIN {X 0,Y 468.828,Z 423.162,A -85,B 0,C 180,E1 -7637.006,E2 -7637.006} C_VEL
LIN {X 0,Y 468.5,Z 431.176,A -85,B 0,C 180,E1 -7637.697,E2 -7637.697} C_VEL
LIN {X 0,Y 468.086,Z 439.29,A -85,B 0,C 180,E1 -7638.525,E2 -7638.525} C_VEL
LIN {X 0,Y 467.722,Z 446.511,A -85,B 0,C 180,E1 -7639.393,E2 -7639.393} C_VEL
LIN {X 0,Y 467.452,Z 452.714,A -85,B 0,C 180,E1 -7640.262,E2 -7640.262} C_VEL
LIN {X 0,Y 467.16,Z 459.251,A -85,B 0,C 180,E1 -7641.348,E2 -7641.348} C_VEL
LIN {X 0,Y 466.98,Z 463.752,A -85,B 0,C 180,E1 -7642.215,E2 -7642.215} C_VEL
LIN {X 0,Y 466.794,Z 469.407,A -85,B 0,C 180,E1 -7643.563,E2 -7643.563} C_VEL
LIN {X 0,Y 466.736,Z 473.565,A -85,B 0,C 180,E1 -7644.816,E2 -7644.816} C_VEL
LIN {X 0,Y 466.648,Z 475.928,A -85,B 0,C 180,E1 -7645.681,E2 -7645.681} C_VEL
LIN {X 0,Y 466.689,Z 477.726,A -85,B 0,C 180,E1 -7646.547,E2 -7646.547} C_VEL
LIN {X 0,Y 466.608,Z 480.165,A -85,B 0,C 180,E1 -7648.274,E2 -7648.274} C_VEL
LIN {X 0,Y 466.619,Z 480.753,A -85,B 0,C 180,E1 -7649.137,E2 -7649.137} C_VEL
LIN {X 0,Y 466.619,Z 480.753,A -85,B 0,C 180,E1 -7650.863,E2 -7650.863} C_VEL
LIN {X 0,Y 466.608,Z 480.165,A -85,B 0,C 180,E1 -7651.726,E2 -7651.726} C_VEL
LIN {X 0,Y 466.689,Z 477.726,A -85,B 0,C 180,E1 -7653.453,E2 -7653.453} C_VEL
LIN {X 0,Y 466.691,Z 474.78,A -85,B 0,C 180,E1 -7654.751,E2 -7654.751} C_VEL
LIN {X 0,Y 466.745,Z 470.795,A -85,B 0,C 180,E1 -7656.05,E2 -7656.05} C_VEL
LIN {X 0,Y 466.869,Z 465.667,A -85,B 0,C 180,E1 -7657.351,E2 -7657.351} C_VEL
LIN {X 0,Y 467.111,Z 460.407,A -85,B 0,C 180,E1 -7658.435,E2 -7658.435} C_VEL
LIN {X 0,Y 467.369,Z 454.09,A -85,B 0,C 180,E1 -7659.521,E2 -7659.521} C_VEL
LIN {X 0,Y 467.607,Z 448.137,A -85,B 0,C 180,E1 -7660.39,E2 -7660.39} C_VEL
LIN {X 0,Y 467.977,Z 441.209,A -85,B 0,C 180,E1 -7661.258,E2 -7661.258} C_VEL
LIN {X 0,Y 468.404,Z 433.029,A -85,B 0,C 180,E1 -7662.126,E2 -7662.126} C_VEL
LIN {X 0,Y 468.738,Z 425.108,A -85,B 0,C 180,E1 -7662.838,E2 -7662.838} C_VEL
LIN {X 0,Y 469.183,Z 415.796,A -85,B 0,C 180,E1 -7663.536,E2 -7663.536} C_VEL
LIN {X 0,Y 469.614,Z 406.035,A -85,B 0,C 180,E1 -7664.13,E2 -7664.13} C_VEL
LIN {X 0,Y 469.919,Z 397.238,A -85,B 0,C 180,E1 -7664.563,E2 -7664.563} C_VEL
LIN {X 0,Y 470.282,Z 387.309,A -85,B 0,C 180,E1 -7664.939,E2 -7664.939} C_VEL
LIN {X 0,Y 470.567,Z 377.453,A -85,B 0,C 180,E1 -7665.206,E2 -7665.206} C_VEL
LIN {X 0,Y 470.808,Z 353.273,A -85,B 0,C 180,E1 -7665.608,E2 -7665.608} C_VEL
LIN {X 0,Y 471.116,Z 288.77,A -85,B 0,C 180,E1 -7666.599,E2 -7666.599} C_VEL
LIN {X 0,Y 467.964,Z 270.237,A -85,B 0,C 180,E1 -7667.023,E2 -7667.023} C_VEL
LIN {X 0,Y 467.929,Z 268.728,A -85,B 0,C 180,E1 -7667.278,E2 -7667.278} C_VEL
LIN {X 0,Y 468.535,Z 255.853,A -85,B 0,C 180,E1 -7670.182,E2 -7670.182} C_VEL
LIN {X 0,Y 469.153,Z 241.253,A -85,B 0,C 180,E1 -7673.389,E2 -7673.389} C_VEL
LIN {X 0,Y 469.408,Z 233.999,A -85,B 0,C 180,E1 -7675.021,E2 -7675.021} C_VEL
LIN {X 0,Y 467.75,Z 224.507,A -85,B 0,C 180,E1 -7677.344,E2 -7677.344} C_VEL
LIN {X 0,Y 467.631,Z 223.754,A -85,B 0,C 180,E1 -7677.608,E2 -7677.608} C_VEL
LIN {X 0,Y 467.57,Z 223.743,A -85,B 0,C 180,E1 -7681.045,E2 -7681.045} C_VEL
LIN {X 0,Y 467.59,Z 223.739,A -85,B 0,C 180,E1 -7684.242,E2 -7684.242} C_VEL
LIN {X 0,Y 467.55,Z 223.742,A -85,B 0,C 180,E1 -7687.186,E2 -7687.186} C_VEL
LIN {X 0,Y 467.579,Z 223.728,A -85,B 0,C 180,E1 -7690.264,E2 -7690.264} C_VEL
LIN {X 0,Y 467.588,Z 223.736,A -85,B 0,C 180,E1 -7692.567,E2 -7692.567} C_VEL
LIN {X 0,Y 467.567,Z 223.739,A -85,B 0,C 180,E1 -7695.052,E2 -7695.052} C_VEL
LIN {X 0,Y 467.59,Z 223.741,A -85,B 0,C 180,E1 -7697.44,E2 -7697.44} C_VEL
LIN {X 0,Y 467.561,Z 223.736,A -85,B 0,C 180,E1 -7700.853,E2 -7700.853} C_VEL
LIN {X 0,Y 467.56,Z 223.737,A -85,B 0,C 180,E1 -7704.261,E2 -7704.261} C_VEL
LIN {X 0,Y 467.574,Z 223.737,A -85,B 0,C 180,E1 -7707.322,E2 -7707.322} C_VEL
LIN {X 0,Y 467.57,Z 223.738,A -85,B 0,C 180,E1 -7710.667,E2 -7710.667} C_VEL
LIN {X 0,Y 467.616,Z 223.726,A -85,B 0,C 180,E1 -7713.199,E2 -7713.199} C_VEL
LIN {X 0,Y 467.593,Z 223.735,A -85,B 0,C 180,E1 -7716.468,E2 -7716.468} C_VEL
LIN {X 0,Y 467.622,Z 223.724,A -85,B 0,C 180,E1 -7719.777,E2 -7719.777} C_VEL
LIN {X 0,Y 467.598,Z 223.724,A -85,B 0,C 180,E1 -7722.506,E2 -7722.506} C_VEL
LIN {X 0,Y 467.606,Z 223.74,A -85,B 0,C 180,E1 -7725.196,E2 -7725.196} C_VEL
LIN {X 0,Y 467.656,Z 223.723,A -85,B 0,C 180,E1 -7727.854,E2 -7727.854} C_VEL
LIN {X 0,Y 467.669,Z 223.72,A -85,B 0,C 180,E1 -7731.357,E2 -7731.357} C_VEL
LIN {X 0,Y 467.723,Z 223.718,A -85,B 0,C 180,E1 -7733.962,E2 -7733.962} C_VEL
LIN {X 0,Y 467.859,Z 223.699,A -85,B 0,C 180,E1 -7737.417,E2 -7737.417} C_VEL
LIN {X 0,Y 467.881,Z 223.684,A -85,B 0,C 180,E1 -7740,E2 -7740} C_VEL
LIN {X 0,Y 467.858,Z 223.699,A -85,B 0,C 180,E1 -7742.582,E2 -7742.582} C_VEL
LIN {X 0,Y 467.734,Z 223.719,A -85,B 0,C 180,E1 -7746.037,E2 -7746.037} C_VEL
LIN {X 0,Y 467.68,Z 223.717,A -85,B 0,C 180,E1 -7748.642,E2 -7748.642} C_VEL
LIN {X 0,Y 467.654,Z 223.723,A -85,B 0,C 180,E1 -7752.145,E2 -7752.145} C_VEL
LIN {X 0,Y 467.638,Z 223.73,A -85,B 0,C 180,E1 -7755.695,E2 -7755.695} C_VEL
LIN {X 0,Y 467.615,Z 223.722,A -85,B 0,C 180,E1 -7758.764,E2 -7758.764} C_VEL
LIN {X 0,Y 467.578,Z 223.734,A -85,B 0,C 180,E1 -7761.268,E2 -7761.268} C_VEL
LIN {X 0,Y 467.56,Z 223.743,A -85,B 0,C 180,E1 -7763.943,E2 -7763.943} C_VEL
LIN {X 0,Y 467.61,Z 223.723,A -85,B 0,C 180,E1 -7766.8,E2 -7766.8} C_VEL
LIN {X 0,Y 467.551,Z 223.74,A -85,B 0,C 180,E1 -7769.738,E2 -7769.738} C_VEL
LIN {X 0,Y 467.58,Z 223.735,A -85,B 0,C 180,E1 -7772.758,E2 -7772.758} C_VEL
LIN {X 0,Y 467.553,Z 223.74,A -85,B 0,C 180,E1 -7775.889,E2 -7775.889} C_VEL
LIN {X 0,Y 467.579,Z 223.737,A -85,B 0,C 180,E1 -7779.144,E2 -7779.144} C_VEL
LIN {X 0,Y 467.616,Z 223.734,A -85,B 0,C 180,E1 -7782.571,E2 -7782.571} C_VEL
LIN {X 0,Y 467.567,Z 223.737,A -85,B 0,C 180,E1 -7785.053,E2 -7785.053} C_VEL
LIN {X 0,Y 467.585,Z 223.721,A -85,B 0,C 180,E1 -7787.44,E2 -7787.44} C_VEL
LIN {X 0,Y 467.596,Z 223.734,A -85,B 0,C 180,E1 -7790.857,E2 -7790.857} C_VEL
LIN {X 0,Y 467.559,Z 223.732,A -85,B 0,C 180,E1 -7794.26,E2 -7794.26} C_VEL
LIN {X 0,Y 467.579,Z 223.738,A -85,B 0,C 180,E1 -7797.321,E2 -7797.321} C_VEL
LIN {X 0,Y 467.566,Z 223.729,A -85,B 0,C 180,E1 -7800.667,E2 -7800.667} C_VEL
LIN {X 0,Y 467.613,Z 223.739,A -85,B 0,C 180,E1 -7803.2,E2 -7803.2} C_VEL
LIN {X 0,Y 467.589,Z 223.738,A -85,B 0,C 180,E1 -7806.468,E2 -7806.468} C_VEL
LIN {X 0,Y 467.62,Z 223.738,A -85,B 0,C 180,E1 -7809.777,E2 -7809.777} C_VEL
LIN {X 0,Y 467.605,Z 223.737,A -85,B 0,C 180,E1 -7812.507,E2 -7812.507} C_VEL
LIN {X 0,Y 467.596,Z 223.74,A -85,B 0,C 180,E1 -7815.422,E2 -7815.422} C_VEL
LIN {X 0,Y 466.925,Z 223.822,A -85,B 0,C 180,E1 -7816.141,E2 -7816.141} C_VEL
LIN {X 0,Y 464.081,Z 224.18,A -85,B 0,C 180,E1 -7817.309,E2 -7817.309} C_VEL
LIN {X 0,Y 461.682,Z 224.477,A -85,B 0,C 180,E1 -7818.251,E2 -7818.251} C_VEL
LIN {X 0,Y 460.656,Z 224.606,A -85,B 0,C 180,E1 -7818.979,E2 -7818.979} C_VEL
LIN {X 0,Y 460.574,Z 224.615,A -85,B 0,C 180,E1 -7819.225,E2 -7819.225} C_VEL
LIN {X 0,Y 460.716,Z 224.598,A -85,B 0,C 180,E1 -7822.538,E2 -7822.538} C_VEL
LIN {X 0,Y 460.696,Z 224.602,A -85,B 0,C 180,E1 -7824.748,E2 -7824.748} C_VEL
LIN {X 0,Y 460.822,Z 224.586,A -85,B 0,C 180,E1 -7827.378,E2 -7827.378} C_VEL
LIN {X 0,Y 460.85,Z 224.58,A -85,B 0,C 180,E1 -7830,E2 -7830} C_VEL
LIN {X 0,Y 460.822,Z 224.586,A -85,B 0,C 180,E1 -7832.622,E2 -7832.622} C_VEL
LIN {X 0,Y 460.709,Z 224.597,A -85,B 0,C 180,E1 -7836.13,E2 -7836.13} C_VEL
LIN {X 0,Y 460.626,Z 224.611,A -85,B 0,C 180,E1 -7838.776,E2 -7838.776} C_VEL
LIN {X 0,Y 460.61,Z 224.612,A -85,B 0,C 180,E1 -7842.445,E2 -7842.445} C_VEL
LIN {X 0,Y 460.596,Z 224.612,A -85,B 0,C 180,E1 -7845.998,E2 -7845.998} C_VEL
LIN {X 0,Y 460.568,Z 224.617,A -85,B 0,C 180,E1 -7848.902,E2 -7848.902} C_VEL
LIN {X 0,Y 460.512,Z 224.62,A -85,B 0,C 180,E1 -7851.486,E2 -7851.486} C_VEL
LIN {X 0,Y 460.538,Z 224.621,A -85,B 0,C 180,E1 -7854.332,E2 -7854.332} C_VEL
LIN {X 0,Y 460.576,Z 224.612,A -85,B 0,C 180,E1 -7857.243,E2 -7857.243} C_VEL
LIN {X 0,Y 460.507,Z 224.613,A -85,B 0,C 180,E1 -7860.24,E2 -7860.24} C_VEL
LIN {X 0,Y 460.526,Z 224.612,A -85,B 0,C 180,E1 -7863.325,E2 -7863.325} C_VEL
LIN {X 0,Y 460.475,Z 224.625,A -85,B 0,C 180,E1 -7866.529,E2 -7866.529} C_VEL
LIN {X 0,Y 460.571,Z 224.61,A -85,B 0,C 180,E1 -7869.858,E2 -7869.858} C_VEL
LIN {X 0,Y 460.509,Z 224.603,A -85,B 0,C 180,E1 -7872.901,E2 -7872.901} C_VEL
LIN {X 0,Y 460.521,Z 224.619,A -85,B 0,C 180,E1 -7875.829,E2 -7875.829} C_VEL
LIN {X 0,Y 460.539,Z 224.608,A -85,B 0,C 180,E1 -7878.99,E2 -7878.99} C_VEL
LIN {X 0,Y 460.536,Z 224.615,A -85,B 0,C 180,E1 -7881.269,E2 -7881.269} C_VEL
LIN {X 0,Y 460.509,Z 224.612,A -85,B 0,C 180,E1 -7884.555,E2 -7884.555} C_VEL
LIN {X 0,Y 460.528,Z 224.619,A -85,B 0,C 180,E1 -7887.716,E2 -7887.716} C_VEL
LIN {X 0,Y 460.537,Z 224.612,A -85,B 0,C 180,E1 -7890.769,E2 -7890.769} C_VEL
LIN {X 0,Y 460.553,Z 224.608,A -85,B 0,C 180,E1 -7893.735,E2 -7893.735} C_VEL
LIN {X 0,Y 460.541,Z 224.614,A -85,B 0,C 180,E1 -7896.624,E2 -7896.624} C_VEL
LIN {X 0,Y 460.549,Z 224.61,A -85,B 0,C 180,E1 -7899.453,E2 -7899.453} C_VEL
LIN {X 0,Y 460.557,Z 224.606,A -85,B 0,C 180,E1 -7902.231,E2 -7902.231} C_VEL
LIN {X 0,Y 460.566,Z 224.612,A -85,B 0,C 180,E1 -7904.965,E2 -7904.965} C_VEL
LIN {X 0,Y 460.61,Z 224.598,A -85,B 0,C 180,E1 -7908.56,E2 -7908.56} C_VEL
LIN {X 0,Y 460.694,Z 224.59,A -85,B 0,C 180,E1 -7912.109,E2 -7912.109} C_VEL
LIN {X 0,Y 460.694,Z 224.596,A -85,B 0,C 180,E1 -7914.749,E2 -7914.749} C_VEL
LIN {X 0,Y 460.823,Z 224.576,A -85,B 0,C 180,E1 -7917.378,E2 -7917.378} C_VEL
LIN {X 0,Y 460.852,Z 224.559,A -85,B 0,C 180,E1 -7920,E2 -7920} C_VEL
LIN {X 0,Y 460.8,Z 224.579,A -85,B 0,C 180,E1 -7922.623,E2 -7922.623} C_VEL
LIN {X 0,Y 460.687,Z 224.594,A -85,B 0,C 180,E1 -7926.131,E2 -7926.131} C_VEL
LIN {X 0,Y 460.619,Z 224.595,A -85,B 0,C 180,E1 -7928.777,E2 -7928.777} C_VEL
LIN {X 0,Y 460.613,Z 224.602,A -85,B 0,C 180,E1 -7932.445,E2 -7932.445} C_VEL
LIN {X 0,Y 460.6,Z 224.603,A -85,B 0,C 180,E1 -7935.998,E2 -7935.998} C_VEL
LIN {X 0,Y 460.568,Z 224.601,A -85,B 0,C 180,E1 -7939.616,E2 -7939.616} C_VEL
LIN {X 0,Y 460.511,Z 224.62,A -85,B 0,C 180,E1 -7942.429,E2 -7942.429} C_VEL
LIN {X 0,Y 460.558,Z 224.605,A -85,B 0,C 180,E1 -7945.8,E2 -7945.8} C_VEL
LIN {X 0,Y 460.553,Z 224.607,A -85,B 0,C 180,E1 -7948.233,E2 -7948.233} C_VEL
LIN {X 0,Y 460.52,Z 224.617,A -85,B 0,C 180,E1 -7951.283,E2 -7951.283} C_VEL
LIN {X 0,Y 460.523,Z 224.612,A -85,B 0,C 180,E1 -7954.504,E2 -7954.504} C_VEL
LIN {X 0,Y 460.502,Z 224.62,A -85,B 0,C 180,E1 -7957.624,E2 -7957.624} C_VEL
LIN {X 0,Y 460.54,Z 224.613,A -85,B 0,C 180,E1 -7960.269,E2 -7960.269} C_VEL
LIN {X 0,Y 460.5,Z 224.619,A -85,B 0,C 180,E1 -7963.376,E2 -7963.376} C_VEL
LIN {X 0,Y 460.5,Z 224.623,A -85,B 0,C 180,E1 -7966.625,E2 -7966.625} C_VEL
LIN {X 0,Y 460.543,Z 224.604,A -85,B 0,C 180,E1 -7969.731,E2 -7969.731} C_VEL
LIN {X 0,Y 460.502,Z 224.622,A -85,B 0,C 180,E1 -7972.524,E2 -7972.524} C_VEL
LIN {X 0,Y 460.548,Z 224.615,A -85,B 0,C 180,E1 -7975.624,E2 -7975.624} C_VEL
LIN {X 0,Y 460.54,Z 224.62,A -85,B 0,C 180,E1 -7978.745,E2 -7978.745} C_VEL
LIN {X 0,Y 460.612,Z 224.72,A -85,B 0,C 180,E1 -7982.248,E2 -7982.248} C_VEL
LIN {X 0,Y 462.11,Z 232.991,A -85,B 0,C 180,E1 -7984.351,E2 -7984.351} C_VEL
LIN {X 0,Y 462.46,Z 236.926,A -85,B 0,C 180,E1 -7985.297,E2 -7985.297} C_VEL
LIN {X 0,Y 461.707,Z 252.374,A -85,B 0,C 180,E1 -7988.807,E2 -7988.807} C_VEL
LIN {X 0,Y 461.141,Z 265.735,A -85,B 0,C 180,E1 -7991.794,E2 -7991.794} C_VEL
LIN {X 0,Y 460.891,Z 269.66,A -85,B 0,C 180,E1 -7992.673,E2 -7992.673} C_VEL
LIN {X 0,Y 461.507,Z 273.104,A -85,B 0,C 180,E1 -7992.8,E2 -7992.8} C_VEL
LIN {X 0,Y 464.368,Z 289.98,A -85,B 0,C 180,E1 -7993.175,E2 -7993.175} C_VEL
LIN {X 0,Y 463.743,Z 374.596,A -85,B 0,C 180,E1 -7994.508,E2 -7994.508} C_VEL
LIN {X 0,Y 463.48,Z 384.493,A -85,B 0,C 180,E1 -7994.752,E2 -7994.752} C_VEL
LIN {X 0,Y 463.17,Z 394.47,A -85,B 0,C 180,E1 -7995.108,E2 -7995.108} C_VEL
LIN {X 0,Y 462.801,Z 403.827,A -85,B 0,C 180,E1 -7995.545,E2 -7995.545} C_VEL
LIN {X 0,Y 462.35,Z 413.97,A -85,B 0,C 180,E1 -7996.148,E2 -7996.148} C_VEL
LIN {X 0,Y 461.89,Z 422.968,A -85,B 0,C 180,E1 -7996.807,E2 -7996.807} C_VEL
LIN {X 0,Y 461.523,Z 431.181,A -85,B 0,C 180,E1 -7997.528,E2 -7997.528} C_VEL
LIN {X 0,Y 461.104,Z 439.097,A -85,B 0,C 180,E1 -7998.349,E2 -7998.349} C_VEL
LIN {X 0,Y 460.711,Z 446.317,A -85,B 0,C 180,E1 -7999.23,E2 -7999.23} C_VEL
LIN {X 0,Y 460.438,Z 452.521,A -85,B 0,C 180,E1 -8000.112,E2 -8000.112} C_VEL
LIN {X 0,Y 460.121,Z 459.058,A -85,B 0,C 180,E1 -8001.214,E2 -8001.214} C_VEL
LIN {X 0,Y 459.901,Z 463.558,A -85,B 0,C 180,E1 -8002.095,E2 -8002.095} C_VEL
LIN {X 0,Y 459.737,Z 468.542,A -85,B 0,C 180,E1 -8003.273,E2 -8003.273} C_VEL
LIN {X 0,Y 459.649,Z 473.372,A -85,B 0,C 180,E1 -8004.736,E2 -8004.736} C_VEL
LIN {X 0,Y 459.566,Z 475.735,A -85,B 0,C 180,E1 -8005.615,E2 -8005.615} C_VEL
LIN {X 0,Y 459.584,Z 477.533,A -85,B 0,C 180,E1 -8006.493,E2 -8006.493} C_VEL
LIN {X 0,Y 459.521,Z 479.973,A -85,B 0,C 180,E1 -8008.247,E2 -8008.247} C_VEL
LIN {X 0,Y 459.522,Z 480.56,A -85,B 0,C 180,E1 -8009.124,E2 -8009.124} C_VEL
LIN {X 0,Y 459.522,Z 480.56,A -85,B 0,C 180,E1 -8010.876,E2 -8010.876} C_VEL
LIN {X 0,Y 459.521,Z 479.973,A -85,B 0,C 180,E1 -8011.753,E2 -8011.753} C_VEL
LIN {X 0,Y 459.584,Z 477.533,A -85,B 0,C 180,E1 -8013.507,E2 -8013.507} C_VEL
LIN {X 0,Y 459.618,Z 474.587,A -85,B 0,C 180,E1 -8014.824,E2 -8014.824} C_VEL
LIN {X 0,Y 459.655,Z 470.601,A -85,B 0,C 180,E1 -8016.144,E2 -8016.144} C_VEL
LIN {X 0,Y 459.814,Z 465.473,A -85,B 0,C 180,E1 -8017.465,E2 -8017.465} C_VEL
LIN {X 0,Y 460.047,Z 460.213,A -85,B 0,C 180,E1 -8018.566,E2 -8018.566} C_VEL
LIN {X 0,Y 460.355,Z 453.896,A -85,B 0,C 180,E1 -8019.668,E2 -8019.668} C_VEL
LIN {X 0,Y 460.59,Z 447.943,A -85,B 0,C 180,E1 -8020.551,E2 -8020.551} C_VEL
LIN {X 0,Y 460.985,Z 441.016,A -85,B 0,C 180,E1 -8021.431,E2 -8021.431} C_VEL
LIN {X 0,Y 461.421,Z 432.835,A -85,B 0,C 180,E1 -8022.312,E2 -8022.312} C_VEL
LIN {X 0,Y 461.828,Z 424.02,A -85,B 0,C 180,E1 -8023.108,E2 -8023.108} C_VEL
LIN {X 0,Y 462.252,Z 415.602,A -85,B 0,C 180,E1 -8023.742,E2 -8023.742} C_VEL
LIN {X 0,Y 462.687,Z 405.841,A -85,B 0,C 180,E1 -8024.346,E2 -8024.346} C_VEL
LIN {X 0,Y 463.1,Z 395.757,A -85,B 0,C 180,E1 -8024.838,E2 -8024.838} C_VEL
LIN {X 0,Y 463.471,Z 386.243,A -85,B 0,C 180,E1 -8025.192,E2 -8025.192} C_VEL
LIN {X 0,Y 463.741,Z 375.929,A -85,B 0,C 180,E1 -8025.464,E2 -8025.464} C_VEL
LIN {X 0,Y 464.329,Z 298.292,A -85,B 0,C 180,E1 -8026.695,E2 -8026.695} C_VEL
LIN {X 0,Y 464.277,Z 289.341,A -85,B 0,C 180,E1 -8026.839,E2 -8026.839} C_VEL
LIN {X 0,Y 460.919,Z 270.107,A -85,B 0,C 180,E1 -8027.287,E2 -8027.287} C_VEL
LIN {X 0,Y 460.933,Z 268.964,A -85,B 0,C 180,E1 -8027.446,E2 -8027.446} C_VEL
LIN {X 0,Y 461.611,Z 255.689,A -85,B 0,C 180,E1 -8030.498,E2 -8030.498} C_VEL
LIN {X 0,Y 462.333,Z 239.645,A -85,B 0,C 180,E1 -8034.09,E2 -8034.09} C_VEL
LIN {X 0,Y 462.405,Z 234.882,A -85,B 0,C 180,E1 -8035.186,E2 -8035.186} C_VEL
LIN {X 0,Y 460.609,Z 224.716,A -85,B 0,C 180,E1 -8037.752,E2 -8037.752} C_VEL
LIN {X 0,Y 460.523,Z 224.622,A -85,B 0,C 180,E1 -8041.283,E2 -8041.283} C_VEL
LIN {X 0,Y 460.534,Z 224.616,A -85,B 0,C 180,E1 -8044.505,E2 -8044.505} C_VEL
LIN {X 0,Y 460.503,Z 224.624,A -85,B 0,C 180,E1 -8047.623,E2 -8047.623} C_VEL
LIN {X 0,Y 460.543,Z 224.604,A -85,B 0,C 180,E1 -8050.269,E2 -8050.269} C_VEL
LIN {X 0,Y 460.5,Z 224.623,A -85,B 0,C 180,E1 -8053.375,E2 -8053.375} C_VEL
LIN {X 0,Y 460.5,Z 224.619,A -85,B 0,C 180,E1 -8056.624,E2 -8056.624} C_VEL
LIN {X 0,Y 460.54,Z 224.613,A -85,B 0,C 180,E1 -8059.731,E2 -8059.731} C_VEL
LIN {X 0,Y 460.5,Z 224.62,A -85,B 0,C 180,E1 -8062.523,E2 -8062.523} C_VEL
LIN {X 0,Y 460.537,Z 224.61,A -85,B 0,C 180,E1 -8065.622,E2 -8065.622} C_VEL
LIN {X 0,Y 460.538,Z 224.615,A -85,B 0,C 180,E1 -8068.744,E2 -8068.744} C_VEL
LIN {X 0,Y 460.582,Z 224.6,A -85,B 0,C 180,E1 -8072.253,E2 -8072.253} C_VEL
LIN {X 0,Y 460.547,Z 224.607,A -85,B 0,C 180,E1 -8074.704,E2 -8074.704} C_VEL
LIN {X 0,Y 460.511,Z 224.62,A -85,B 0,C 180,E1 -8077.571,E2 -8077.571} C_VEL
LIN {X 0,Y 460.568,Z 224.601,A -85,B 0,C 180,E1 -8080.384,E2 -8080.384} C_VEL
LIN {X 0,Y 460.604,Z 224.603,A -85,B 0,C 180,E1 -8084.059,E2 -8084.059} C_VEL
LIN {X 0,Y 460.609,Z 224.601,A -85,B 0,C 180,E1 -8087.665,E2 -8087.665} C_VEL
LIN {X 0,Y 460.619,Z 224.595,A -85,B 0,C 180,E1 -8091.223,E2 -8091.223} C_VEL
LIN {X 0,Y 460.687,Z 224.594,A -85,B 0,C 180,E1 -8093.869,E2 -8093.869} C_VEL
LIN {X 0,Y 460.8,Z 224.579,A -85,B 0,C 180,E1 -8097.377,E2 -8097.377} C_VEL
LIN {X 0,Y 460.852,Z 224.559,A -85,B 0,C 180,E1 -8100,E2 -8100} C_VEL
LIN {X 0,Y 460.823,Z 224.576,A -85,B 0,C 180,E1 -8102.622,E2 -8102.622} C_VEL
LIN {X 0,Y 460.701,Z 224.596,A -85,B 0,C 180,E1 -8106.13,E2 -8106.13} C_VEL
LIN {X 0,Y 460.627,Z 224.593,A -85,B 0,C 180,E1 -8108.776,E2 -8108.776} C_VEL
LIN {X 0,Y 460.612,Z 224.604,A -85,B 0,C 180,E1 -8112.444,E2 -8112.444} C_VEL
LIN {X 0,Y 460.598,Z 224.609,A -85,B 0,C 180,E1 -8115.997,E2 -8115.997} C_VEL
LIN {X 0,Y 460.568,Z 224.598,A -85,B 0,C 180,E1 -8118.901,E2 -8118.901} C_VEL
LIN {X 0,Y 460.513,Z 224.614,A -85,B 0,C 180,E1 -8121.485,E2 -8121.485} C_VEL
LIN {X 0,Y 460.528,Z 224.621,A -85,B 0,C 180,E1 -8124.332,E2 -8124.332} C_VEL
LIN {X 0,Y 460.568,Z 224.597,A -85,B 0,C 180,E1 -8127.243,E2 -8127.243} C_VEL
LIN {X 0,Y 460.508,Z 224.624,A -85,B 0,C 180,E1 -8130.24,E2 -8130.24} C_VEL
LIN {X 0,Y 460.526,Z 224.613,A -85,B 0,C 180,E1 -8133.324,E2 -8133.324} C_VEL
LIN {X 0,Y 460.475,Z 224.625,A -85,B 0,C 180,E1 -8136.529,E2 -8136.529} C_VEL
LIN {X 0,Y 460.555,Z 224.613,A -85,B 0,C 180,E1 -8139.859,E2 -8139.859} C_VEL
LIN {X 0,Y 460.539,Z 224.615,A -85,B 0,C 180,E1 -8142.904,E2 -8142.904} C_VEL
LIN {X 0,Y 460.508,Z 224.612,A -85,B 0,C 180,E1 -8145.83,E2 -8145.83} C_VEL
LIN {X 0,Y 460.535,Z 224.6,A -85,B 0,C 180,E1 -8148.989,E2 -8148.989} C_VEL
LIN {X 0,Y 460.536,Z 224.616,A -85,B 0,C 180,E1 -8151.268,E2 -8151.268} C_VEL
LIN {X 0,Y 460.509,Z 224.608,A -85,B 0,C 180,E1 -8154.554,E2 -8154.554} C_VEL
LIN {X 0,Y 460.529,Z 224.622,A -85,B 0,C 180,E1 -8157.716,E2 -8157.716} C_VEL
LIN {X 0,Y 460.536,Z 224.605,A -85,B 0,C 180,E1 -8160.769,E2 -8160.769} C_VEL
LIN {X 0,Y 460.559,Z 224.618,A -85,B 0,C 180,E1 -8163.735,E2 -8163.735} C_VEL
LIN {X 0,Y 460.542,Z 224.617,A -85,B 0,C 180,E1 -8166.624,E2 -8166.624} C_VEL
LIN {X 0,Y 460.549,Z 224.621,A -85,B 0,C 180,E1 -8169.453,E2 -8169.453} C_VEL
LIN {X 0,Y 460.556,Z 224.616,A -85,B 0,C 180,E1 -8172.23,E2 -8172.23} C_VEL
LIN {X 0,Y 460.564,Z 224.617,A -85,B 0,C 180,E1 -8174.965,E2 -8174.965} C_VEL
LIN {X 0,Y 460.608,Z 224.61,A -85,B 0,C 180,E1 -8178.559,E2 -8178.559} C_VEL
LIN {X 0,Y 460.574,Z 224.615,A -85,B 0,C 180,E1 -8179.225,E2 -8179.225} C_VEL
LIN {X 0,Y 459.92,Z 224.7,A -85,B 0,C 180,E1 -8179.955,E2 -8179.955} C_VEL
LIN {X 0,Y 457.102,Z 225.055,A -85,B 0,C 180,E1 -8181.142,E2 -8181.142} C_VEL
LIN {X 0,Y 454.722,Z 225.349,A -85,B 0,C 180,E1 -8182.099,E2 -8182.099} C_VEL
LIN {X 0,Y 453.711,Z 225.471,A -85,B 0,C 180,E1 -8182.838,E2 -8182.838} C_VEL
LIN {X 0,Y 453.634,Z 225.48,A -85,B 0,C 180,E1 -8183.088,E2 -8183.088} C_VEL
LIN {X 0,Y 453.67,Z 225.477,A -85,B 0,C 180,E1 -8184.667,E2 -8184.667} C_VEL
LIN {X 0,Y 453.762,Z 225.465,A -85,B 0,C 180,E1 -8187.337,E2 -8187.337} C_VEL
LIN {X 0,Y 453.821,Z 225.456,A -85,B 0,C 180,E1 -8190,E2 -8190} C_VEL
LIN {X 0,Y 453.762,Z 225.465,A -85,B 0,C 180,E1 -8192.663,E2 -8192.663} C_VEL
LIN {X 0,Y 453.676,Z 225.474,A -85,B 0,C 180,E1 -8196.225,E2 -8196.225} C_VEL
LIN {X 0,Y 453.589,Z 225.487,A -85,B 0,C 180,E1 -8198.913,E2 -8198.913} C_VEL
LIN {X 0,Y 453.56,Z 225.49,A -85,B 0,C 180,E1 -8202.529,E2 -8202.529} C_VEL
LIN {X 0,Y 453.541,Z 225.491,A -85,B 0,C 180,E1 -8206.196,E2 -8206.196} C_VEL
LIN {X 0,Y 453.517,Z 225.495,A -85,B 0,C 180,E1 -8209.041,E2 -8209.041} C_VEL
LIN {X 0,Y 453.472,Z 225.498,A -85,B 0,C 180,E1 -8211.836,E2 -8211.836} C_VEL
LIN {X 0,Y 453.51,Z 225.496,A -85,B 0,C 180,E1 -8214.735,E2 -8214.735} C_VEL
LIN {X 0,Y 453.534,Z 225.491,A -85,B 0,C 180,E1 -8217.961,E2 -8217.961} C_VEL
LIN {X 0,Y 453.463,Z 225.497,A -85,B 0,C 180,E1 -8221.526,E2 -8221.526} C_VEL
LIN {X 0,Y 453.485,Z 225.482,A -85,B 0,C 180,E1 -8224.778,E2 -8224.778} C_VEL
LIN {X 0,Y 453.477,Z 225.5,A -85,B 0,C 180,E1 -8228.31,E2 -8228.31} C_VEL
LIN {X 0,Y 453.512,Z 225.476,A -85,B 0,C 180,E1 -8230.607,E2 -8230.607} C_VEL
LIN {X 0,Y 453.462,Z 225.49,A -85,B 0,C 180,E1 -8234.221,E2 -8234.221} C_VEL
LIN {X 0,Y 453.488,Z 225.493,A -85,B 0,C 180,E1 -8237.009,E2 -8237.009} C_VEL
LIN {X 0,Y 453.525,Z 225.489,A -85,B 0,C 180,E1 -8240.555,E2 -8240.555} C_VEL
LIN {X 0,Y 453.453,Z 225.498,A -85,B 0,C 180,E1 -8243.918,E2 -8243.918} C_VEL
LIN {X 0,Y 453.48,Z 225.491,A -85,B 0,C 180,E1 -8247.152,E2 -8247.152} C_VEL
LIN {X 0,Y 453.472,Z 225.494,A -85,B 0,C 180,E1 -8250.269,E2 -8250.269} C_VEL
LIN {X 0,Y 453.498,Z 225.48,A -85,B 0,C 180,E1 -8253.294,E2 -8253.294} C_VEL
LIN {X 0,Y 453.494,Z 225.494,A -85,B 0,C 180,E1 -8256.239,E2 -8256.239} C_VEL
LIN {X 0,Y 453.48,Z 225.492,A -85,B 0,C 180,E1 -8259.118,E2 -8259.118} C_VEL
LIN {X 0,Y 453.51,Z 225.486,A -85,B 0,C 180,E1 -8261.945,E2 -8261.945} C_VEL
LIN {X 0,Y 453.539,Z 225.486,A -85,B 0,C 180,E1 -8264.727,E2 -8264.727} C_VEL
LIN {X 0,Y 453.558,Z 225.476,A -85,B 0,C 180,E1 -8268.379,E2 -8268.379} C_VEL
LIN {X 0,Y 453.651,Z 225.468,A -85,B 0,C 180,E1 -8271.986,E2 -8271.986} C_VEL
LIN {X 0,Y 453.667,Z 225.471,A -85,B 0,C 180,E1 -8274.667,E2 -8274.667} C_VEL
LIN {X 0,Y 453.763,Z 225.456,A -85,B 0,C 180,E1 -8277.337,E2 -8277.337} C_VEL
LIN {X 0,Y 453.822,Z 225.434,A -85,B 0,C 180,E1 -8280,E2 -8280} C_VEL
LIN {X 0,Y 453.744,Z 225.458,A -85,B 0,C 180,E1 -8282.664,E2 -8282.664} C_VEL
LIN {X 0,Y 453.653,Z 225.471,A -85,B 0,C 180,E1 -8286.226,E2 -8286.226} C_VEL
LIN {X 0,Y 453.585,Z 225.469,A -85,B 0,C 180,E1 -8288.914,E2 -8288.914} C_VEL
LIN {X 0,Y 453.563,Z 225.48,A -85,B 0,C 180,E1 -8292.529,E2 -8292.529} C_VEL
LIN {X 0,Y 453.544,Z 225.483,A -85,B 0,C 180,E1 -8296.196,E2 -8296.196} C_VEL
LIN {X 0,Y 453.517,Z 225.479,A -85,B 0,C 180,E1 -8299.04,E2 -8299.04} C_VEL
LIN {X 0,Y 453.477,Z 225.492,A -85,B 0,C 180,E1 -8301.837,E2 -8301.837} C_VEL
LIN {X 0,Y 453.508,Z 225.49,A -85,B 0,C 180,E1 -8304.735,E2 -8304.735} C_VEL
LIN {X 0,Y 453.533,Z 225.479,A -85,B 0,C 180,E1 -8307.96,E2 -8307.96} C_VEL
LIN {X 0,Y 453.464,Z 225.495,A -85,B 0,C 180,E1 -8311.525,E2 -8311.525} C_VEL
LIN {X 0,Y 453.483,Z 225.491,A -85,B 0,C 180,E1 -8314.777,E2 -8314.777} C_VEL
LIN {X 0,Y 453.461,Z 225.502,A -85,B 0,C 180,E1 -8318.312,E2 -8318.312} C_VEL
LIN {X 0,Y 453.495,Z 225.493,A -85,B 0,C 180,E1 -8320.609,E2 -8320.609} C_VEL
LIN {X 0,Y 453.456,Z 225.496,A -85,B 0,C 180,E1 -8323.244,E2 -8323.244} C_VEL
LIN {X 0,Y 453.465,Z 225.497,A -85,B 0,C 180,E1 -8325.779,E2 -8325.779} C_VEL
LIN {X 0,Y 453.481,Z 225.491,A -85,B 0,C 180,E1 -8328.21,E2 -8328.21} C_VEL
LIN {X 0,Y 453.512,Z 225.49,A -85,B 0,C 180,E1 -8330.791,E2 -8330.791} C_VEL
LIN {X 0,Y 453.456,Z 225.495,A -85,B 0,C 180,E1 -8333.918,E2 -8333.918} C_VEL
LIN {X 0,Y 453.485,Z 225.493,A -85,B 0,C 180,E1 -8337.152,E2 -8337.152} C_VEL
LIN {X 0,Y 453.469,Z 225.496,A -85,B 0,C 180,E1 -8340.268,E2 -8340.268} C_VEL
LIN {X 0,Y 453.557,Z 225.626,A -85,B 0,C 180,E1 -8342.035,E2 -8342.035} C_VEL
LIN {X 0,Y 455.223,Z 234.741,A -85,B 0,C 180,E1 -8344.388,E2 -8344.388} C_VEL
LIN {X 0,Y 455.451,Z 238.741,A -85,B 0,C 180,E1 -8345.378,E2 -8345.378} C_VEL
LIN {X 0,Y 454.65,Z 254.275,A -85,B 0,C 180,E1 -8348.937,E2 -8348.937} C_VEL
LIN {X 0,Y 454.021,Z 267.49,A -85,B 0,C 180,E1 -8351.966,E2 -8351.966} C_VEL
LIN {X 0,Y 453.922,Z 269.472,A -85,B 0,C 180,E1 -8352.398,E2 -8352.398} C_VEL
LIN {X 0,Y 454.427,Z 272.786,A -85,B 0,C 180,E1 -8352.522,E2 -8352.522} C_VEL
LIN {X 0,Y 457.564,Z 291.078,A -85,B 0,C 180,E1 -8352.938,E2 -8352.938} C_VEL
LIN {X 0,Y 456.903,Z 374.404,A -85,B 0,C 180,E1 -8354.27,E2 -8354.27} C_VEL
LIN {X 0,Y 456.643,Z 384.3,A -85,B 0,C 180,E1 -8354.518,E2 -8354.518} C_VEL
LIN {X 0,Y 456.31,Z 394.277,A -85,B 0,C 180,E1 -8354.879,E2 -8354.879} C_VEL
LIN {X 0,Y 455.895,Z 403.633,A -85,B 0,C 180,E1 -8355.321,E2 -8355.321} C_VEL
LIN {X 0,Y 455.428,Z 413.777,A -85,B 0,C 180,E1 -8355.934,E2 -8355.934} C_VEL
LIN {X 0,Y 454.97,Z 422.775,A -85,B 0,C 180,E1 -8356.602,E2 -8356.602} C_VEL
LIN {X 0,Y 454.556,Z 431.184,A -85,B 0,C 180,E1 -8357.353,E2 -8357.353} C_VEL
LIN {X 0,Y 454.127,Z 438.903,A -85,B 0,C 180,E1 -8358.167,E2 -8358.167} C_VEL
LIN {X 0,Y 453.682,Z 446.123,A -85,B 0,C 180,E1 -8359.061,E2 -8359.061} C_VEL
LIN {X 0,Y 453.411,Z 452.327,A -85,B 0,C 180,E1 -8359.958,E2 -8359.958} C_VEL
LIN {X 0,Y 453.048,Z 458.864,A -85,B 0,C 180,E1 -8361.076,E2 -8361.076} C_VEL
LIN {X 0,Y 452.849,Z 463.365,A -85,B 0,C 180,E1 -8361.971,E2 -8361.971} C_VEL
LIN {X 0,Y 452.645,Z 469.011,A -85,B 0,C 180,E1 -8363.358,E2 -8363.358} C_VEL
LIN {X 0,Y 452.562,Z 473.178,A -85,B 0,C 180,E1 -8364.654,E2 -8364.654} C_VEL
LIN {X 0,Y 452.488,Z 475.542,A -85,B 0,C 180,E1 -8365.546,E2 -8365.546} C_VEL
LIN {X 0,Y 452.481,Z 477.339,A -85,B 0,C 180,E1 -8366.438,E2 -8366.438} C_VEL
LIN {X 0,Y 452.437,Z 479.78,A -85,B 0,C 180,E1 -8368.22,E2 -8368.22} C_VEL
LIN {X 0,Y 452.429,Z 480.367,A -85,B 0,C 180,E1 -8369.11,E2 -8369.11} C_VEL
LIN {X 0,Y 452.429,Z 480.367,A -85,B 0,C 180,E1 -8370.89,E2 -8370.89} C_VEL
LIN {X 0,Y 452.437,Z 479.78,A -85,B 0,C 180,E1 -8371.78,E2 -8371.78} C_VEL
LIN {X 0,Y 452.481,Z 477.339,A -85,B 0,C 180,E1 -8373.562,E2 -8373.562} C_VEL
LIN {X 0,Y 452.546,Z 474.395,A -85,B 0,C 180,E1 -8374.9,E2 -8374.9} C_VEL
LIN {X 0,Y 452.585,Z 470.408,A -85,B 0,C 180,E1 -8376.24,E2 -8376.24} C_VEL
LIN {X 0,Y 452.74,Z 465.28,A -85,B 0,C 180,E1 -8377.582,E2 -8377.582} C_VEL
LIN {X 0,Y 453.007,Z 460.02,A -85,B 0,C 180,E1 -8378.7,E2 -8378.7} C_VEL
LIN {X 0,Y 453.327,Z 453.703,A -85,B 0,C 180,E1 -8379.819,E2 -8379.819} C_VEL
LIN {X 0,Y 453.582,Z 447.749,A -85,B 0,C 180,E1 -8380.716,E2 -8380.716} C_VEL
LIN {X 0,Y 454,Z 440.822,A -85,B 0,C 180,E1 -8381.61,E2 -8381.61} C_VEL
LIN {X 0,Y 454.451,Z 432.641,A -85,B 0,C 180,E1 -8382.504,E2 -8382.504} C_VEL
LIN {X 0,Y 454.866,Z 424.625,A -85,B 0,C 180,E1 -8383.245,E2 -8383.245} C_VEL
LIN {X 0,Y 455.34,Z 415.409,A -85,B 0,C 180,E1 -8383.955,E2 -8383.955} C_VEL
LIN {X 0,Y 455.809,Z 405.648,A -85,B 0,C 180,E1 -8384.567,E2 -8384.567} C_VEL
LIN {X 0,Y 456.182,Z 396.852,A -85,B 0,C 180,E1 -8385.012,E2 -8385.012} C_VEL
LIN {X 0,Y 456.61,Z 386.924,A -85,B 0,C 180,E1 -8385.397,E2 -8385.397} C_VEL
LIN {X 0,Y 456.888,Z 377.068,A -85,B 0,C 180,E1 -8385.673,E2 -8385.673} C_VEL
LIN {X 0,Y 457.161,Z 351.802,A -85,B 0,C 180,E1 -8386.103,E2 -8386.103} C_VEL
LIN {X 0,Y 457.504,Z 290.456,A -85,B 0,C 180,E1 -8387.074,E2 -8387.074} C_VEL
LIN {X 0,Y 453.935,Z 269.713,A -85,B 0,C 180,E1 -8387.575,E2 -8387.575} C_VEL
LIN {X 0,Y 453.967,Z 268.438,A -85,B 0,C 180,E1 -8387.805,E2 -8387.805} C_VEL
LIN {X 0,Y 454.646,Z 255.524,A -85,B 0,C 180,E1 -8390.826,E2 -8390.826} C_VEL
LIN {X 0,Y 455.354,Z 241.386,A -85,B 0,C 180,E1 -8394.049,E2 -8394.049} C_VEL
LIN {X 0,Y 455.387,Z 235.766,A -85,B 0,C 180,E1 -8395.357,E2 -8395.357} C_VEL
LIN {X 0,Y 453.745,Z 226.589,A -85,B 0,C 180,E1 -8397.688,E2 -8397.688} C_VEL
LIN {X 0,Y 453.541,Z 225.496,A -85,B 0,C 180,E1 -8398.081,E2 -8398.081} C_VEL
LIN {X 0,Y 453.468,Z 225.501,A -85,B 0,C 180,E1 -8401.525,E2 -8401.525} C_VEL
LIN {X 0,Y 453.489,Z 225.492,A -85,B 0,C 180,E1 -8404.777,E2 -8404.777} C_VEL
LIN {X 0,Y 453.467,Z 225.497,A -85,B 0,C 180,E1 -8408.311,E2 -8408.311} C_VEL
LIN {X 0,Y 453.496,Z 225.48,A -85,B 0,C 180,E1 -8410.609,E2 -8410.609} C_VEL
LIN {X 0,Y 453.456,Z 225.499,A -85,B 0,C 180,E1 -8413.244,E2 -8413.244} C_VEL
